LIN {X 0,Y 523.96,Z 722.024,A -85,B 0,C 180,E1 -4662.837,E2 -4662.837} C_VEL
LIN {X 0,Y 524.007,Z 722.026,A -85,B 0,C 180,E1 -4665.236,E2 -4665.236} C_VEL
LIN {X 0,Y 524.015,Z 722.018,A -85,B 0,C 180,E1 -4668.394,E2 -4668.394} C_VEL
LIN {X 0,Y 524.003,Z 722.019,A -85,B 0,C 180,E1 -4671.516,E2 -4671.516} C_VEL
LIN {X 0,Y 524.085,Z 722.007,A -85,B 0,C 180,E1 -4674.614,E2 -4674.614} C_VEL
LIN {X 0,Y 524.116,Z 722.011,A -85,B 0,C 180,E1 -4677.694,E2 -4677.694} C_VEL
LIN {X 0,Y 524.126,Z 722.001,A -85,B 0,C 180,E1 -4680.768,E2 -4680.768} C_VEL
LIN {X 0,Y 524.075,Z 722.005,A -85,B 0,C 180,E1 -4683.075,E2 -4683.075} C_VEL
LIN {X 0,Y 524.046,Z 722.017,A -85,B 0,C 180,E1 -4686.159,E2 -4686.159} C_VEL
LIN {X 0,Y 524.002,Z 722.022,A -85,B 0,C 180,E1 -4689.262,E2 -4689.262} C_VEL
LIN {X 0,Y 524.005,Z 722.021,A -85,B 0,C 180,E1 -4691.739,E2 -4691.739} C_VEL
LIN {X 0,Y 523.995,Z 722.019,A -85,B 0,C 180,E1 -4695.052,E2 -4695.052} C_VEL
LIN {X 0,Y 523.967,Z 722.031,A -85,B 0,C 180,E1 -4697.969,E2 -4697.969} C_VEL
LIN {X 0,Y 523.974,Z 722.02,A -85,B 0,C 180,E1 -4700.41,E2 -4700.41} C_VEL
LIN {X 0,Y 523.919,Z 722.028,A -85,B 0,C 180,E1 -4702.893,E2 -4702.893} C_VEL
LIN {X 0,Y 523.955,Z 722.027,A -85,B 0,C 180,E1 -4705.418,E2 -4705.418} C_VEL
LIN {X 0,Y 523.972,Z 722.031,A -85,B 0,C 180,E1 -4707.999,E2 -4707.999} C_VEL
LIN {X 0,Y 523.947,Z 722.026,A -85,B 0,C 180,E1 -4710.855,E2 -4710.855} C_VEL
LIN {X 0,Y 523.963,Z 722.028,A -85,B 0,C 180,E1 -4713.735,E2 -4713.735} C_VEL
LIN {X 0,Y 523.925,Z 722.029,A -85,B 0,C 180,E1 -4716.404,E2 -4716.404} C_VEL
LIN {X 0,Y 523.933,Z 722.012,A -85,B 0,C 180,E1 -4719.084,E2 -4719.084} C_VEL
LIN {X 0,Y 523.974,Z 722.017,A -85,B 0,C 180,E1 -4721.312,E2 -4721.312} C_VEL
LIN {X 0,Y 523.957,Z 722.031,A -85,B 0,C 180,E1 -4724.691,E2 -4724.691} C_VEL
LIN {X 0,Y 523.958,Z 722.023,A -85,B 0,C 180,E1 -4727.882,E2 -4727.882} C_VEL
LIN {X 0,Y 523.928,Z 722.034,A -85,B 0,C 180,E1 -4730.916,E2 -4730.916} C_VEL
LIN {X 0,Y 523.929,Z 722.027,A -85,B 0,C 180,E1 -4733.828,E2 -4733.828} C_VEL
LIN {X 0,Y 523.945,Z 722.036,A -85,B 0,C 180,E1 -4736.636,E2 -4736.636} C_VEL
LIN {X 0,Y 523.958,Z 722.022,A -85,B 0,C 180,E1 -4739.356,E2 -4739.356} C_VEL
LIN {X 0,Y 523.979,Z 722.027,A -85,B 0,C 180,E1 -4742.281,E2 -4742.281} C_VEL
LIN {X 0,Y 523.949,Z 722.033,A -85,B 0,C 180,E1 -4744.581,E2 -4744.581} C_VEL
LIN {X 0,Y 523.97,Z 722.172,A -85,B 0,C 180,E1 -4747.4,E2 -4747.4} C_VEL
LIN {X 0,Y 524.887,Z 728.251,A -85,B 0,C 180,E1 -4748.601,E2 -4748.601} C_VEL
LIN {X 0,Y 524.571,Z 744.644,A -85,B 0,C 180,E1 -4751.649,E2 -4751.649} C_VEL
LIN {X 0,Y 524.221,Z 761.458,A -85,B 0,C 180,E1 -4754.724,E2 -4754.724} C_VEL
LIN {X 0,Y 523.899,Z 779.887,A -85,B 0,C 180,E1 -4758.045,E2 -4758.045} C_VEL
LIN {X 0,Y 524.091,Z 781.846,A -85,B 0,C 180,E1 -4758.12,E2 -4758.12} C_VEL
LIN {X 0,Y 524.986,Z 790.156,A -85,B 0,C 180,E1 -4758.254,E2 -4758.254} C_VEL
LIN {X 0,Y 524.799,Z 856.138,A -85,B 0,C 180,E1 -4759.17,E2 -4759.17} C_VEL
LIN {X 0,Y 524.675,Z 865.409,A -85,B 0,C 180,E1 -4759.387,E2 -4759.387} C_VEL
LIN {X 0,Y 524.58,Z 873.883,A -85,B 0,C 180,E1 -4759.677,E2 -4759.677} C_VEL
LIN {X 0,Y 524.407,Z 882.388,A -85,B 0,C 180,E1 -4760.064,E2 -4760.064} C_VEL
LIN {X 0,Y 524.242,Z 890.722,A -85,B 0,C 180,E1 -4760.548,E2 -4760.548} C_VEL
LIN {X 0,Y 524.079,Z 898.761,A -85,B 0,C 180,E1 -4761.129,E2 -4761.129} C_VEL
LIN {X 0,Y 523.896,Z 907.432,A -85,B 0,C 180,E1 -4761.903,E2 -4761.903} C_VEL
LIN {X 0,Y 523.734,Z 915.938,A -85,B 0,C 180,E1 -4762.87,E2 -4762.87} C_VEL
LIN {X 0,Y 523.637,Z 922.61,A -85,B 0,C 180,E1 -4763.836,E2 -4763.836} C_VEL
LIN {X 0,Y 523.484,Z 926.989,A -85,B 0,C 180,E1 -4764.607,E2 -4764.607} C_VEL
LIN {X 0,Y 523.469,Z 932.149,A -85,B 0,C 180,E1 -4765.765,E2 -4765.765} C_VEL
LIN {X 0,Y 523.38,Z 935.937,A -85,B 0,C 180,E1 -4766.921,E2 -4766.921} C_VEL
LIN {X 0,Y 523.334,Z 937.681,A -85,B 0,C 180,E1 -4767.691,E2 -4767.691} C_VEL
LIN {X 0,Y 523.273,Z 938.93,A -85,B 0,C 180,E1 -4768.461,E2 -4768.461} C_VEL
LIN {X 0,Y 523.248,Z 939.707,A -85,B 0,C 180,E1 -4769.23,E2 -4769.23} C_VEL
LIN {X 0,Y 523.244,Z 940,A -85,B 0,C 180,E1 -4770,E2 -4770} C_VEL
LIN {X 0,Y 523.248,Z 939.707,A -85,B 0,C 180,E1 -4770.77,E2 -4770.77} C_VEL
LIN {X 0,Y 523.273,Z 938.929,A -85,B 0,C 180,E1 -4771.539,E2 -4771.539} C_VEL
LIN {X 0,Y 523.334,Z 937.68,A -85,B 0,C 180,E1 -4772.309,E2 -4772.309} C_VEL
LIN {X 0,Y 523.407,Z 934.786,A -85,B 0,C 180,E1 -4773.464,E2 -4773.464} C_VEL
LIN {X 0,Y 523.469,Z 932.149,A -85,B 0,C 180,E1 -4774.235,E2 -4774.235} C_VEL
LIN {X 0,Y 523.484,Z 926.986,A -85,B 0,C 180,E1 -4775.393,E2 -4775.393} C_VEL
LIN {X 0,Y 523.668,Z 920.738,A -85,B 0,C 180,E1 -4776.468,E2 -4776.468} C_VEL
LIN {X 0,Y 523.757,Z 912.74,A -85,B 0,C 180,E1 -4777.518,E2 -4777.518} C_VEL
LIN {X 0,Y 523.931,Z 905.398,A -85,B 0,C 180,E1 -4778.291,E2 -4778.291} C_VEL
LIN {X 0,Y 524.102,Z 897.534,A -85,B 0,C 180,E1 -4778.968,E2 -4778.968} C_VEL
LIN {X 0,Y 524.272,Z 889.222,A -85,B 0,C 180,E1 -4779.549,E2 -4779.549} C_VEL
LIN {X 0,Y 524.477,Z 878.61,A -85,B 0,C 180,E1 -4780.13,E2 -4780.13} C_VEL
LIN {X 0,Y 524.667,Z 867.075,A -85,B 0,C 180,E1 -4780.565,E2 -4780.565} C_VEL
LIN {X 0,Y 524.763,Z 857.437,A -85,B 0,C 180,E1 -4780.807,E2 -4780.807} C_VEL
LIN {X 0,Y 524.938,Z 807.339,A -85,B 0,C 180,E1 -4781.512,E2 -4781.512} C_VEL
LIN {X 0,Y 524.813,Z 787.359,A -85,B 0,C 180,E1 -4781.788,E2 -4781.788} C_VEL
LIN {X 0,Y 523.904,Z 780.121,A -85,B 0,C 180,E1 -4781.935,E2 -4781.935} C_VEL
LIN {X 0,Y 523.982,Z 772.996,A -85,B 0,C 180,E1 -4783.18,E2 -4783.18} C_VEL
LIN {X 0,Y 524.271,Z 757.745,A -85,B 0,C 180,E1 -4785.951,E2 -4785.951} C_VEL
LIN {X 0,Y 524.624,Z 741.367,A -85,B 0,C 180,E1 -4788.957,E2 -4788.957} C_VEL
LIN {X 0,Y 524.887,Z 728.251,A -85,B 0,C 180,E1 -4791.399,E2 -4791.399} C_VEL
LIN {X 0,Y 523.952,Z 722.075,A -85,B 0,C 180,E1 -4792.643,E2 -4792.643} C_VEL
LIN {X 0,Y 523.949,Z 722.033,A -85,B 0,C 180,E1 -4795.419,E2 -4795.419} C_VEL
LIN {X 0,Y 523.97,Z 722.026,A -85,B 0,C 180,E1 -4797.999,E2 -4797.999} C_VEL
LIN {X 0,Y 523.948,Z 722.024,A -85,B 0,C 180,E1 -4800.855,E2 -4800.855} C_VEL
LIN {X 0,Y 523.963,Z 722.03,A -85,B 0,C 180,E1 -4803.735,E2 -4803.735} C_VEL
LIN {X 0,Y 523.924,Z 722.028,A -85,B 0,C 180,E1 -4806.404,E2 -4806.404} C_VEL
LIN {X 0,Y 523.928,Z 722.033,A -85,B 0,C 180,E1 -4809.084,E2 -4809.084} C_VEL
LIN {X 0,Y 523.958,Z 722.024,A -85,B 0,C 180,E1 -4812.118,E2 -4812.118} C_VEL
LIN {X 0,Y 523.957,Z 722.031,A -85,B 0,C 180,E1 -4815.309,E2 -4815.309} C_VEL
LIN {X 0,Y 523.974,Z 722.016,A -85,B 0,C 180,E1 -4818.688,E2 -4818.688} C_VEL
LIN {X 0,Y 523.927,Z 722.013,A -85,B 0,C 180,E1 -4821.079,E2 -4821.079} C_VEL
LIN {X 0,Y 523.93,Z 722.033,A -85,B 0,C 180,E1 -4823.828,E2 -4823.828} C_VEL
LIN {X 0,Y 523.944,Z 722.028,A -85,B 0,C 180,E1 -4826.636,E2 -4826.636} C_VEL
LIN {X 0,Y 523.958,Z 722.026,A -85,B 0,C 180,E1 -4829.356,E2 -4829.356} C_VEL
LIN {X 0,Y 523.981,Z 722.026,A -85,B 0,C 180,E1 -4832.281,E2 -4832.281} C_VEL
LIN {X 0,Y 523.955,Z 722.027,A -85,B 0,C 180,E1 -4834.582,E2 -4834.582} C_VEL
LIN {X 0,Y 523.919,Z 722.027,A -85,B 0,C 180,E1 -4837.107,E2 -4837.107} C_VEL
LIN {X 0,Y 523.981,Z 722.023,A -85,B 0,C 180,E1 -4839.866,E2 -4839.866} C_VEL
LIN {X 0,Y 523.973,Z 722.024,A -85,B 0,C 180,E1 -4842.838,E2 -4842.838} C_VEL
LIN {X 0,Y 523.979,Z 722.021,A -85,B 0,C 180,E1 -4845.236,E2 -4845.236} C_VEL
LIN {X 0,Y 524.015,Z 722.021,A -85,B 0,C 180,E1 -4848.394,E2 -4848.394} C_VEL
LIN {X 0,Y 524.007,Z 722.019,A -85,B 0,C 180,E1 -4851.516,E2 -4851.516} C_VEL
LIN {X 0,Y 524.084,Z 722.013,A -85,B 0,C 180,E1 -4854.614,E2 -4854.614} C_VEL
LIN {X 0,Y 524.114,Z 721.998,A -85,B 0,C 180,E1 -4857.695,E2 -4857.695} C_VEL
LIN {X 0,Y 524.126,Z 722.01,A -85,B 0,C 180,E1 -4860.768,E2 -4860.768} C_VEL
LIN {X 0,Y 524.075,Z 722.013,A -85,B 0,C 180,E1 -4863.075,E2 -4863.075} C_VEL
LIN {X 0,Y 524.04,Z 722.015,A -85,B 0,C 180,E1 -4866.159,E2 -4866.159} C_VEL
LIN {X 0,Y 524.003,Z 722.018,A -85,B 0,C 180,E1 -4868.484,E2 -4868.484} C_VEL
LIN {X 0,Y 524.006,Z 722.019,A -85,B 0,C 180,E1 -4871.74,E2 -4871.74} C_VEL
LIN {X 0,Y 523.996,Z 722.023,A -85,B 0,C 180,E1 -4875.052,E2 -4875.052} C_VEL
LIN {X 0,Y 523.95,Z 722.021,A -85,B 0,C 180,E1 -4877.97,E2 -4877.97} C_VEL
LIN {X 0,Y 523.974,Z 722.024,A -85,B 0,C 180,E1 -4880.41,E2 -4880.41} C_VEL
LIN {X 0,Y 523.912,Z 722.04,A -85,B 0,C 180,E1 -4882.894,E2 -4882.894} C_VEL
LIN {X 0,Y 523.985,Z 722.016,A -85,B 0,C 180,E1 -4886.019,E2 -4886.019} C_VEL
LIN {X 0,Y 523.937,Z 722.033,A -85,B 0,C 180,E1 -4888.875,E2 -4888.875} C_VEL
LIN {X 0,Y 523.921,Z 722.032,A -85,B 0,C 180,E1 -4891.544,E2 -4891.544} C_VEL
LIN {X 0,Y 523.922,Z 722.027,A -85,B 0,C 180,E1 -4894.291,E2 -4894.291} C_VEL
LIN {X 0,Y 523.908,Z 722.039,A -85,B 0,C 180,E1 -4897.132,E2 -4897.132} C_VEL
LIN {X 0,Y 523.939,Z 722.023,A -85,B 0,C 180,E1 -4900.13,E2 -4900.13} C_VEL
LIN {X 0,Y 523.933,Z 722.013,A -85,B 0,C 180,E1 -4902.458,E2 -4902.458} C_VEL
LIN {X 0,Y 523.944,Z 722.029,A -85,B 0,C 180,E1 -4905.31,E2 -4905.31} C_VEL
LIN {X 0,Y 523.916,Z 722.032,A -85,B 0,C 180,E1 -4906.909,E2 -4906.909} C_VEL
LIN {X 0,Y 523.252,Z 722.122,A -85,B 0,C 180,E1 -4907.55,E2 -4907.55} C_VEL
LIN {X 0,Y 520.412,Z 722.471,A -85,B 0,C 180,E1 -4908.592,E2 -4908.592} C_VEL
LIN {X 0,Y 518.007,Z 722.774,A -85,B 0,C 180,E1 -4909.431,E2 -4909.431} C_VEL
LIN {X 0,Y 516.97,Z 722.894,A -85,B 0,C 180,E1 -4910.079,E2 -4910.079} C_VEL
LIN {X 0,Y 516.883,Z 722.903,A -85,B 0,C 180,E1 -4910.298,E2 -4910.298} C_VEL
LIN {X 0,Y 516.878,Z 722.909,A -85,B 0,C 180,E1 -4913.343,E2 -4913.343} C_VEL
LIN {X 0,Y 516.885,Z 722.909,A -85,B 0,C 180,E1 -4916.119,E2 -4916.119} C_VEL
LIN {X 0,Y 516.891,Z 722.903,A -85,B 0,C 180,E1 -4918.936,E2 -4918.936} C_VEL
LIN {X 0,Y 516.864,Z 722.917,A -85,B 0,C 180,E1 -4921.581,E2 -4921.581} C_VEL
LIN {X 0,Y 516.885,Z 722.911,A -85,B 0,C 180,E1 -4924.208,E2 -4924.208} C_VEL
LIN {X 0,Y 516.86,Z 722.909,A -85,B 0,C 180,E1 -4926.776,E2 -4926.776} C_VEL
LIN {X 0,Y 516.941,Z 722.908,A -85,B 0,C 180,E1 -4929.732,E2 -4929.732} C_VEL
LIN {X 0,Y 517.031,Z 723.121,A -85,B 0,C 180,E1 -4931.32,E2 -4931.32} C_VEL
LIN {X 0,Y 517.103,Z 730.186,A -85,B 0,C 180,E1 -4933.01,E2 -4933.01} C_VEL
LIN {X 0,Y 516.819,Z 742.298,A -85,B 0,C 180,E1 -4935.831,E2 -4935.831} C_VEL
LIN {X 0,Y 516.707,Z 751.608,A -85,B 0,C 180,E1 -4937.94,E2 -4937.94} C_VEL
LIN {X 0,Y 517.044,Z 754.054,A -85,B 0,C 180,E1 -4938.029,E2 -4938.029} C_VEL
LIN {X 0,Y 518.001,Z 762.348,A -85,B 0,C 180,E1 -4938.167,E2 -4938.167} C_VEL
LIN {X 0,Y 517.785,Z 826.462,A -85,B 0,C 180,E1 -4939.07,E2 -4939.07} C_VEL
LIN {X 0,Y 517.706,Z 835.644,A -85,B 0,C 180,E1 -4939.292,E2 -4939.292} C_VEL
LIN {X 0,Y 517.546,Z 845.274,A -85,B 0,C 180,E1 -4939.634,E2 -4939.634} C_VEL
LIN {X 0,Y 517.414,Z 855.328,A -85,B 0,C 180,E1 -4940.126,E2 -4940.126} C_VEL
LIN {X 0,Y 517.184,Z 865.799,A -85,B 0,C 180,E1 -4940.812,E2 -4940.812} C_VEL
LIN {X 0,Y 516.898,Z 875.032,A -85,B 0,C 180,E1 -4941.595,E2 -4941.595} C_VEL
LIN {X 0,Y 516.703,Z 882.414,A -85,B 0,C 180,E1 -4942.379,E2 -4942.379} C_VEL
LIN {X 0,Y 516.597,Z 889.273,A -85,B 0,C 180,E1 -4943.277,E2 -4943.277} C_VEL
LIN {X 0,Y 516.499,Z 895.801,A -85,B 0,C 180,E1 -4944.339,E2 -4944.339} C_VEL
LIN {X 0,Y 516.322,Z 900.458,A -85,B 0,C 180,E1 -4945.315,E2 -4945.315} C_VEL
LIN {X 0,Y 516.385,Z 903.47,A -85,B 0,C 180,E1 -4946.098,E2 -4946.098} C_VEL
LIN {X 0,Y 516.295,Z 905.809,A -85,B 0,C 180,E1 -4946.879,E2 -4946.879} C_VEL
LIN {X 0,Y 516.263,Z 907.59,A -85,B 0,C 180,E1 -4947.659,E2 -4947.659} C_VEL
LIN {X 0,Y 516.19,Z 908.875,A -85,B 0,C 180,E1 -4948.44,E2 -4948.44} C_VEL
LIN {X 0,Y 516.157,Z 909.689,A -85,B 0,C 180,E1 -4949.22,E2 -4949.22} C_VEL
LIN {X 0,Y 516.152,Z 909.997,A -85,B 0,C 180,E1 -4950,E2 -4950} C_VEL
LIN {X 0,Y 516.157,Z 909.726,A -85,B 0,C 180,E1 -4950.78,E2 -4950.78} C_VEL
LIN {X 0,Y 516.191,Z 908.986,A -85,B 0,C 180,E1 -4951.56,E2 -4951.56} C_VEL
LIN {X 0,Y 516.263,Z 907.777,A -85,B 0,C 180,E1 -4952.341,E2 -4952.341} C_VEL
LIN {X 0,Y 516.324,Z 904.921,A -85,B 0,C 180,E1 -4953.512,E2 -4953.512} C_VEL
LIN {X 0,Y 516.39,Z 902.325,A -85,B 0,C 180,E1 -4954.293,E2 -4954.293} C_VEL
LIN {X 0,Y 516.431,Z 897.208,A -85,B 0,C 180,E1 -4955.466,E2 -4955.466} C_VEL
LIN {X 0,Y 516.59,Z 891.595,A -85,B 0,C 180,E1 -4956.462,E2 -4956.462} C_VEL
LIN {X 0,Y 516.691,Z 883.161,A -85,B 0,C 180,E1 -4957.621,E2 -4957.621} C_VEL
LIN {X 0,Y 516.916,Z 874.939,A -85,B 0,C 180,E1 -4958.503,E2 -4958.503} C_VEL
LIN {X 0,Y 517.157,Z 865.674,A -85,B 0,C 180,E1 -4959.287,E2 -4959.287} C_VEL
LIN {X 0,Y 517.369,Z 855.163,A -85,B 0,C 180,E1 -4959.974,E2 -4959.974} C_VEL
LIN {X 0,Y 517.578,Z 845.055,A -85,B 0,C 180,E1 -4960.464,E2 -4960.464} C_VEL
LIN {X 0,Y 517.691,Z 836.176,A -85,B 0,C 180,E1 -4960.783,E2 -4960.783} C_VEL
LIN {X 0,Y 517.845,Z 827.357,A -85,B 0,C 180,E1 -4961.001,E2 -4961.001} C_VEL
LIN {X 0,Y 517.932,Z 760.029,A -85,B 0,C 180,E1 -4961.957,E2 -4961.957} C_VEL
LIN {X 0,Y 516.695,Z 751.778,A -85,B 0,C 180,E1 -4962.126,E2 -4962.126} C_VEL
LIN {X 0,Y 516.647,Z 751.291,A -85,B 0,C 180,E1 -4962.172,E2 -4962.172} C_VEL
LIN {X 0,Y 516.952,Z 737.395,A -85,B 0,C 180,E1 -4965.394,E2 -4965.394} C_VEL
LIN {X 0,Y 517.152,Z 725.401,A -85,B 0,C 180,E1 -4968.214,E2 -4968.214} C_VEL
LIN {X 0,Y 516.985,Z 722.989,A -85,B 0,C 180,E1 -4968.836,E2 -4968.836} C_VEL
LIN {X 0,Y 516.887,Z 722.909,A -85,B 0,C 180,E1 -4971.538,E2 -4971.538} C_VEL
LIN {X 0,Y 516.876,Z 722.917,A -85,B 0,C 180,E1 -4974.355,E2 -4974.355} C_VEL
LIN {X 0,Y 516.892,Z 722.907,A -85,B 0,C 180,E1 -4977.535,E2 -4977.535} C_VEL
LIN {X 0,Y 516.888,Z 722.914,A -85,B 0,C 180,E1 -4980.204,E2 -4980.204} C_VEL
LIN {X 0,Y 516.882,Z 722.909,A -85,B 0,C 180,E1 -4982.948,E2 -4982.948} C_VEL
LIN {X 0,Y 516.872,Z 722.911,A -85,B 0,C 180,E1 -4985.78,E2 -4985.78} C_VEL
LIN {X 0,Y 516.879,Z 722.908,A -85,B 0,C 180,E1 -4988.716,E2 -4988.716} C_VEL
LIN {X 0,Y 516.913,Z 722.903,A -85,B 0,C 180,E1 -4991.775,E2 -4991.775} C_VEL
LIN {X 0,Y 516.896,Z 722.903,A -85,B 0,C 180,E1 -4995.007,E2 -4995.007} C_VEL
LIN {X 0,Y 516.914,Z 722.891,A -85,B 0,C 180,E1 -4998.399,E2 -4998.399} C_VEL
LIN {X 0,Y 516.88,Z 722.908,A -85,B 0,C 180,E1 -5001.284,E2 -5001.284} C_VEL
LIN {X 0,Y 516.872,Z 722.91,A -85,B 0,C 180,E1 -5004.22,E2 -5004.22} C_VEL
LIN {X 0,Y 516.883,Z 722.911,A -85,B 0,C 180,E1 -5007.052,E2 -5007.052} C_VEL
LIN {X 0,Y 516.888,Z 722.906,A -85,B 0,C 180,E1 -5009.796,E2 -5009.796} C_VEL
LIN {X 0,Y 516.926,Z 722.903,A -85,B 0,C 180,E1 -5012.467,E2 -5012.467} C_VEL
LIN {X 0,Y 516.908,Z 722.907,A -85,B 0,C 180,E1 -5015.072,E2 -5015.072} C_VEL
LIN {X 0,Y 516.888,Z 722.907,A -85,B 0,C 180,E1 -5018.462,E2 -5018.462} C_VEL
LIN {X 0,Y 516.903,Z 722.91,A -85,B 0,C 180,E1 -5020.955,E2 -5020.955} C_VEL
LIN {X 0,Y 516.911,Z 722.905,A -85,B 0,C 180,E1 -5023.41,E2 -5023.41} C_VEL
LIN {X 0,Y 516.907,Z 722.905,A -85,B 0,C 180,E1 -5025.834,E2 -5025.834} C_VEL
LIN {X 0,Y 516.954,Z 722.903,A -85,B 0,C 180,E1 -5029.028,E2 -5029.028} C_VEL
LIN {X 0,Y 516.98,Z 722.886,A -85,B 0,C 180,E1 -5032.187,E2 -5032.187} C_VEL
LIN {X 0,Y 517.031,Z 722.885,A -85,B 0,C 180,E1 -5034.54,E2 -5034.54} C_VEL
LIN {X 0,Y 517.088,Z 722.887,A -85,B 0,C 180,E1 -5037.663,E2 -5037.663} C_VEL
LIN {X 0,Y 517.096,Z 722.877,A -85,B 0,C 180,E1 -5040.779,E2 -5040.779} C_VEL
LIN {X 0,Y 517.015,Z 722.884,A -85,B 0,C 180,E1 -5043.117,E2 -5043.117} C_VEL
LIN {X 0,Y 517.011,Z 722.892,A -85,B 0,C 180,E1 -5046.243,E2 -5046.243} C_VEL
LIN {X 0,Y 516.956,Z 722.902,A -85,B 0,C 180,E1 -5049.389,E2 -5049.389} C_VEL
LIN {X 0,Y 516.954,Z 722.898,A -85,B 0,C 180,E1 -5051.807,E2 -5051.807} C_VEL
LIN {X 0,Y 516.947,Z 722.898,A -85,B 0,C 180,E1 -5055.146,E2 -5055.146} C_VEL
LIN {X 0,Y 516.928,Z 722.904,A -85,B 0,C 180,E1 -5058.222,E2 -5058.222} C_VEL
LIN {X 0,Y 516.915,Z 722.897,A -85,B 0,C 180,E1 -5060.701,E2 -5060.701} C_VEL
LIN {X 0,Y 516.913,Z 722.912,A -85,B 0,C 180,E1 -5064.072,E2 -5064.072} C_VEL
LIN {X 0,Y 516.928,Z 722.902,A -85,B 0,C 180,E1 -5066.658,E2 -5066.658} C_VEL
LIN {X 0,Y 516.913,Z 722.899,A -85,B 0,C 180,E1 -5069.524,E2 -5069.524} C_VEL
LIN {X 0,Y 516.899,Z 722.909,A -85,B 0,C 180,E1 -5072.544,E2 -5072.544} C_VEL
LIN {X 0,Y 516.885,Z 722.905,A -85,B 0,C 180,E1 -5075.332,E2 -5075.332} C_VEL
LIN {X 0,Y 516.883,Z 722.903,A -85,B 0,C 180,E1 -5077.943,E2 -5077.943} C_VEL
LIN {X 0,Y 516.905,Z 722.9,A -85,B 0,C 180,E1 -5080.739,E2 -5080.739} C_VEL
LIN {X 0,Y 516.884,Z 722.908,A -85,B 0,C 180,E1 -5083.903,E2 -5083.903} C_VEL
LIN {X 0,Y 516.883,Z 722.911,A -85,B 0,C 180,E1 -5086.107,E2 -5086.107} C_VEL
LIN {X 0,Y 516.918,Z 722.904,A -85,B 0,C 180,E1 -5088.398,E2 -5088.398} C_VEL
LIN {X 0,Y 516.886,Z 722.908,A -85,B 0,C 180,E1 -5091.284,E2 -5091.284} C_VEL
LIN {X 0,Y 516.892,Z 722.907,A -85,B 0,C 180,E1 -5094.221,E2 -5094.221} C_VEL
LIN {X 0,Y 516.899,Z 722.907,A -85,B 0,C 180,E1 -5097.053,E2 -5097.053} C_VEL
LIN {X 0,Y 516.894,Z 722.9,A -85,B 0,C 180,E1 -5099.796,E2 -5099.796} C_VEL
LIN {X 0,Y 516.929,Z 722.908,A -85,B 0,C 180,E1 -5102.467,E2 -5102.467} C_VEL
LIN {X 0,Y 516.905,Z 722.909,A -85,B 0,C 180,E1 -5105.072,E2 -5105.072} C_VEL
LIN {X 0,Y 516.908,Z 723.029,A -85,B 0,C 180,E1 -5107.26,E2 -5107.26} C_VEL
LIN {X 0,Y 517.89,Z 729.171,A -85,B 0,C 180,E1 -5108.506,E2 -5108.506} C_VEL
LIN {X 0,Y 517.556,Z 745.565,A -85,B 0,C 180,E1 -5111.596,E2 -5111.596} C_VEL
LIN {X 0,Y 517.158,Z 762.669,A -85,B 0,C 180,E1 -5114.767,E2 -5114.767} C_VEL
LIN {X 0,Y 516.825,Z 779.847,A -85,B 0,C 180,E1 -5117.883,E2 -5117.883} C_VEL
LIN {X 0,Y 517.051,Z 781.622,A -85,B 0,C 180,E1 -5117.954,E2 -5117.954} C_VEL
LIN {X 0,Y 518.035,Z 790.103,A -85,B 0,C 180,E1 -5118.094,E2 -5118.094} C_VEL
LIN {X 0,Y 517.842,Z 856.135,A -85,B 0,C 180,E1 -5119.022,E2 -5119.022} C_VEL
LIN {X 0,Y 517.684,Z 865.407,A -85,B 0,C 180,E1 -5119.242,E2 -5119.242} C_VEL
LIN {X 0,Y 517.604,Z 873.881,A -85,B 0,C 180,E1 -5119.537,E2 -5119.537} C_VEL
LIN {X 0,Y 517.419,Z 882.386,A -85,B 0,C 180,E1 -5119.928,E2 -5119.928} C_VEL
LIN {X 0,Y 517.249,Z 890.72,A -85,B 0,C 180,E1 -5120.419,E2 -5120.419} C_VEL
LIN {X 0,Y 517.068,Z 898.758,A -85,B 0,C 180,E1 -5121.007,E2 -5121.007} C_VEL
LIN {X 0,Y 516.847,Z 907.431,A -85,B 0,C 180,E1 -5121.791,E2 -5121.791} C_VEL
LIN {X 0,Y 516.692,Z 915.938,A -85,B 0,C 180,E1 -5122.772,E2 -5122.772} C_VEL
LIN {X 0,Y 516.571,Z 922.609,A -85,B 0,C 180,E1 -5123.751,E2 -5123.751} C_VEL
LIN {X 0,Y 516.431,Z 926.989,A -85,B 0,C 180,E1 -5124.534,E2 -5124.534} C_VEL
LIN {X 0,Y 516.392,Z 932.149,A -85,B 0,C 180,E1 -5125.707,E2 -5125.707} C_VEL
LIN {X 0,Y 516.325,Z 934.787,A -85,B 0,C 180,E1 -5126.488,E2 -5126.488} C_VEL
LIN {X 0,Y 516.261,Z 937.68,A -85,B 0,C 180,E1 -5127.659,E2 -5127.659} C_VEL
LIN {X 0,Y 516.19,Z 938.929,A -85,B 0,C 180,E1 -5128.44,E2 -5128.44} C_VEL
LIN {X 0,Y 516.158,Z 939.706,A -85,B 0,C 180,E1 -5129.22,E2 -5129.22} C_VEL
LIN {X 0,Y 516.151,Z 940,A -85,B 0,C 180,E1 -5130,E2 -5130} C_VEL
LIN {X 0,Y 516.158,Z 939.706,A -85,B 0,C 180,E1 -5130.78,E2 -5130.78} C_VEL
LIN {X 0,Y 516.19,Z 938.928,A -85,B 0,C 180,E1 -5131.56,E2 -5131.56} C_VEL
LIN {X 0,Y 516.261,Z 937.679,A -85,B 0,C 180,E1 -5132.341,E2 -5132.341} C_VEL
LIN {X 0,Y 516.325,Z 934.786,A -85,B 0,C 180,E1 -5133.512,E2 -5133.512} C_VEL
LIN {X 0,Y 516.392,Z 932.149,A -85,B 0,C 180,E1 -5134.293,E2 -5134.293} C_VEL
LIN {X 0,Y 516.431,Z 926.985,A -85,B 0,C 180,E1 -5135.466,E2 -5135.466} C_VEL
LIN {X 0,Y 516.58,Z 921.233,A -85,B 0,C 180,E1 -5136.478,E2 -5136.478} C_VEL
LIN {X 0,Y 516.686,Z 914.435,A -85,B 0,C 180,E1 -5137.425,E2 -5137.425} C_VEL
LIN {X 0,Y 516.863,Z 906.418,A -85,B 0,C 180,E1 -5138.307,E2 -5138.307} C_VEL
LIN {X 0,Y 517.068,Z 898.763,A -85,B 0,C 180,E1 -5138.993,E2 -5138.993} C_VEL
LIN {X 0,Y 517.249,Z 890.721,A -85,B 0,C 180,E1 -5139.581,E2 -5139.581} C_VEL
LIN {X 0,Y 517.419,Z 882.388,A -85,B 0,C 180,E1 -5140.072,E2 -5140.072} C_VEL
LIN {X 0,Y 517.614,Z 873.885,A -85,B 0,C 180,E1 -5140.463,E2 -5140.463} C_VEL
LIN {X 0,Y 517.71,Z 863.745,A -85,B 0,C 180,E1 -5140.807,E2 -5140.807} C_VEL
LIN {X 0,Y 517.912,Z 852.082,A -85,B 0,C 180,E1 -5141.05,E2 -5141.05} C_VEL
LIN {X 0,Y 517.876,Z 787.906,A -85,B 0,C 180,E1 -5141.94,E2 -5141.94} C_VEL
LIN {X 0,Y 516.843,Z 780.138,A -85,B 0,C 180,E1 -5142.094,E2 -5142.094} C_VEL
LIN {X 0,Y 516.863,Z 777.221,A -85,B 0,C 180,E1 -5142.566,E2 -5142.566} C_VEL
LIN {X 0,Y 517.174,Z 761.553,A -85,B 0,C 180,E1 -5145.437,E2 -5145.437} C_VEL
LIN {X 0,Y 517.556,Z 745.56,A -85,B 0,C 180,E1 -5148.404,E2 -5148.404} C_VEL
LIN {X 0,Y 517.912,Z 730.264,A -85,B 0,C 180,E1 -5151.284,E2 -5151.284} C_VEL
LIN {X 0,Y 517.164,Z 724.233,A -85,B 0,C 180,E1 -5152.469,E2 -5152.469} C_VEL
LIN {X 0,Y 516.905,Z 722.934,A -85,B 0,C 180,E1 -5152.798,E2 -5152.798} C_VEL
LIN {X 0,Y 516.944,Z 722.899,A -85,B 0,C 180,E1 -5156.196,E2 -5156.196} C_VEL
LIN {X 0,Y 516.923,Z 722.906,A -85,B 0,C 180,E1 -5159.304,E2 -5159.304} C_VEL
LIN {X 0,Y 516.902,Z 722.904,A -85,B 0,C 180,E1 -5162.544,E2 -5162.544} C_VEL
LIN {X 0,Y 516.884,Z 722.913,A -85,B 0,C 180,E1 -5165.333,E2 -5165.333} C_VEL
LIN {X 0,Y 516.883,Z 722.91,A -85,B 0,C 180,E1 -5167.943,E2 -5167.943} C_VEL
LIN {X 0,Y 516.887,Z 722.903,A -85,B 0,C 180,E1 -5170.741,E2 -5170.741} C_VEL
LIN {X 0,Y 516.885,Z 722.904,A -85,B 0,C 180,E1 -5172.831,E2 -5172.831} C_VEL
LIN {X 0,Y 516.924,Z 722.904,A -85,B 0,C 180,E1 -5175.01,E2 -5175.01} C_VEL
LIN {X 0,Y 516.924,Z 722.895,A -85,B 0,C 180,E1 -5178.398,E2 -5178.398} C_VEL
LIN {X 0,Y 516.888,Z 722.89,A -85,B 0,C 180,E1 -5181.285,E2 -5181.285} C_VEL
LIN {X 0,Y 516.893,Z 722.907,A -85,B 0,C 180,E1 -5184.221,E2 -5184.221} C_VEL
LIN {X 0,Y 516.898,Z 722.906,A -85,B 0,C 180,E1 -5187.053,E2 -5187.053} C_VEL
LIN {X 0,Y 516.894,Z 722.91,A -85,B 0,C 180,E1 -5189.797,E2 -5189.797} C_VEL
LIN {X 0,Y 516.93,Z 722.903,A -85,B 0,C 180,E1 -5192.468,E2 -5192.468} C_VEL
LIN {X 0,Y 516.913,Z 722.903,A -85,B 0,C 180,E1 -5195.072,E2 -5195.072} C_VEL
LIN {X 0,Y 516.872,Z 722.908,A -85,B 0,C 180,E1 -5197.622,E2 -5197.622} C_VEL
LIN {X 0,Y 516.935,Z 722.905,A -85,B 0,C 180,E1 -5200.13,E2 -5200.13} C_VEL
LIN {X 0,Y 516.933,Z 722.904,A -85,B 0,C 180,E1 -5202.596,E2 -5202.596} C_VEL
LIN {X 0,Y 516.944,Z 722.897,A -85,B 0,C 180,E1 -5205.03,E2 -5205.03} C_VEL
LIN {X 0,Y 516.968,Z 722.897,A -85,B 0,C 180,E1 -5208.234,E2 -5208.234} C_VEL
LIN {X 0,Y 516.972,Z 722.895,A -85,B 0,C 180,E1 -5211.4,E2 -5211.4} C_VEL
LIN {X 0,Y 517.011,Z 722.892,A -85,B 0,C 180,E1 -5213.757,E2 -5213.757} C_VEL
LIN {X 0,Y 517.087,Z 722.873,A -85,B 0,C 180,E1 -5217.663,E2 -5217.663} C_VEL
LIN {X 0,Y 517.096,Z 722.885,A -85,B 0,C 180,E1 -5220.779,E2 -5220.779} C_VEL
LIN {X 0,Y 517.016,Z 722.892,A -85,B 0,C 180,E1 -5223.117,E2 -5223.117} C_VEL
LIN {X 0,Y 517.005,Z 722.892,A -85,B 0,C 180,E1 -5226.243,E2 -5226.243} C_VEL
LIN {X 0,Y 516.948,Z 722.897,A -85,B 0,C 180,E1 -5229.389,E2 -5229.389} C_VEL
LIN {X 0,Y 516.955,Z 722.898,A -85,B 0,C 180,E1 -5231.807,E2 -5231.807} C_VEL
LIN {X 0,Y 516.947,Z 722.899,A -85,B 0,C 180,E1 -5235.147,E2 -5235.147} C_VEL
LIN {X 0,Y 516.918,Z 722.897,A -85,B 0,C 180,E1 -5238.223,E2 -5238.223} C_VEL
LIN {X 0,Y 516.915,Z 722.907,A -85,B 0,C 180,E1 -5240.701,E2 -5240.701} C_VEL
LIN {X 0,Y 516.892,Z 722.904,A -85,B 0,C 180,E1 -5244.073,E2 -5244.073} C_VEL
LIN {X 0,Y 516.926,Z 722.898,A -85,B 0,C 180,E1 -5246.658,E2 -5246.658} C_VEL
LIN {X 0,Y 516.911,Z 722.907,A -85,B 0,C 180,E1 -5249.523,E2 -5249.523} C_VEL
LIN {X 0,Y 516.896,Z 722.904,A -85,B 0,C 180,E1 -5252.543,E2 -5252.543} C_VEL
LIN {X 0,Y 516.867,Z 722.917,A -85,B 0,C 180,E1 -5255.33,E2 -5255.33} C_VEL
LIN {X 0,Y 516.88,Z 722.907,A -85,B 0,C 180,E1 -5257.943,E2 -5257.943} C_VEL
LIN {X 0,Y 516.885,Z 722.902,A -85,B 0,C 180,E1 -5260.742,E2 -5260.742} C_VEL
LIN {X 0,Y 516.864,Z 722.894,A -85,B 0,C 180,E1 -5262.834,E2 -5262.834} C_VEL
LIN {X 0,Y 516.896,Z 722.902,A -85,B 0,C 180,E1 -5265.007,E2 -5265.007} C_VEL
LIN {X 0,Y 516.914,Z 722.903,A -85,B 0,C 180,E1 -5268.399,E2 -5268.399} C_VEL
LIN {X 0,Y 516.883,Z 722.903,A -85,B 0,C 180,E1 -5270.298,E2 -5270.298} C_VEL
LIN {X 0,Y 516.211,Z 722.988,A -85,B 0,C 180,E1 -5270.948,E2 -5270.948} C_VEL
LIN {X 0,Y 513.364,Z 723.349,A -85,B 0,C 180,E1 -5272.004,E2 -5272.004} C_VEL
LIN {X 0,Y 510.955,Z 723.654,A -85,B 0,C 180,E1 -5272.854,E2 -5272.854} C_VEL
LIN {X 0,Y 509.912,Z 723.782,A -85,B 0,C 180,E1 -5273.51,E2 -5273.51} C_VEL
LIN {X 0,Y 509.822,Z 723.792,A -85,B 0,C 180,E1 -5273.733,E2 -5273.733} C_VEL
LIN {X 0,Y 509.843,Z 723.784,A -85,B 0,C 180,E1 -5276.538,E2 -5276.538} C_VEL
LIN {X 0,Y 509.844,Z 723.784,A -85,B 0,C 180,E1 -5279.334,E2 -5279.334} C_VEL
LIN {X 0,Y 509.849,Z 723.789,A -85,B 0,C 180,E1 -5282.052,E2 -5282.052} C_VEL
LIN {X 0,Y 509.813,Z 723.789,A -85,B 0,C 180,E1 -5284.701,E2 -5284.701} C_VEL
LIN {X 0,Y 509.827,Z 723.789,A -85,B 0,C 180,E1 -5287.458,E2 -5287.458} C_VEL
LIN {X 0,Y 509.893,Z 723.786,A -85,B 0,C 180,E1 -5290.683,E2 -5290.683} C_VEL
LIN {X 0,Y 509.996,Z 723.933,A -85,B 0,C 180,E1 -5291.209,E2 -5291.209} C_VEL
LIN {X 0,Y 510.117,Z 730.352,A -85,B 0,C 180,E1 -5292.77,E2 -5292.77} C_VEL
LIN {X 0,Y 509.817,Z 742.464,A -85,B 0,C 180,E1 -5295.633,E2 -5295.633} C_VEL
LIN {X 0,Y 509.675,Z 751.798,A -85,B 0,C 180,E1 -5297.771,E2 -5297.771} C_VEL
LIN {X 0,Y 510.018,Z 754.22,A -85,B 0,C 180,E1 -5297.86,E2 -5297.86} C_VEL
LIN {X 0,Y 511.07,Z 762.602,A -85,B 0,C 180,E1 -5298.005,E2 -5298.005} C_VEL
LIN {X 0,Y 510.838,Z 826.703,A -85,B 0,C 180,E1 -5298.92,E2 -5298.92} C_VEL
LIN {X 0,Y 510.757,Z 835.873,A -85,B 0,C 180,E1 -5299.144,E2 -5299.144} C_VEL
LIN {X 0,Y 510.571,Z 845.496,A -85,B 0,C 180,E1 -5299.491,E2 -5299.491} C_VEL
LIN {X 0,Y 510.423,Z 855.546,A -85,B 0,C 180,E1 -5299.989,E2 -5299.989} C_VEL
LIN {X 0,Y 510.183,Z 865.972,A -85,B 0,C 180,E1 -5300.685,E2 -5300.685} C_VEL
LIN {X 0,Y 509.923,Z 874.121,A -85,B 0,C 180,E1 -5301.38,E2 -5301.38} C_VEL
LIN {X 0,Y 509.713,Z 880.841,A -85,B 0,C 180,E1 -5302.075,E2 -5302.075} C_VEL
LIN {X 0,Y 509.609,Z 887.199,A -85,B 0,C 180,E1 -5302.87,E2 -5302.87} C_VEL
LIN {X 0,Y 509.522,Z 892.483,A -85,B 0,C 180,E1 -5303.665,E2 -5303.665} C_VEL
LIN {X 0,Y 509.385,Z 896.896,A -85,B 0,C 180,E1 -5304.458,E2 -5304.458} C_VEL
LIN {X 0,Y 509.235,Z 900.571,A -85,B 0,C 180,E1 -5305.25,E2 -5305.25} C_VEL
LIN {X 0,Y 509.318,Z 903.564,A -85,B 0,C 180,E1 -5306.044,E2 -5306.044} C_VEL
LIN {X 0,Y 509.213,Z 905.893,A -85,B 0,C 180,E1 -5306.835,E2 -5306.835} C_VEL
LIN {X 0,Y 509.192,Z 907.664,A -85,B 0,C 180,E1 -5307.627,E2 -5307.627} C_VEL
LIN {X 0,Y 509.111,Z 908.944,A -85,B 0,C 180,E1 -5308.418,E2 -5308.418} C_VEL
LIN {X 0,Y 509.07,Z 909.754,A -85,B 0,C 180,E1 -5309.209,E2 -5309.209} C_VEL
LIN {X 0,Y 509.063,Z 910.061,A -85,B 0,C 180,E1 -5310,E2 -5310} C_VEL
LIN {X 0,Y 509.071,Z 909.79,A -85,B 0,C 180,E1 -5310.791,E2 -5310.791} C_VEL
LIN {X 0,Y 509.112,Z 909.052,A -85,B 0,C 180,E1 -5311.582,E2 -5311.582} C_VEL
LIN {X 0,Y 509.192,Z 907.847,A -85,B 0,C 180,E1 -5312.373,E2 -5312.373} C_VEL
LIN {X 0,Y 509.246,Z 905.005,A -85,B 0,C 180,E1 -5313.561,E2 -5313.561} C_VEL
LIN {X 0,Y 509.312,Z 902.421,A -85,B 0,C 180,E1 -5314.353,E2 -5314.353} C_VEL
LIN {X 0,Y 509.378,Z 897.328,A -85,B 0,C 180,E1 -5315.542,E2 -5315.542} C_VEL
LIN {X 0,Y 509.524,Z 892.227,A -85,B 0,C 180,E1 -5316.469,E2 -5316.469} C_VEL
LIN {X 0,Y 509.651,Z 884.971,A -85,B 0,C 180,E1 -5317.528,E2 -5317.528} C_VEL
LIN {X 0,Y 509.876,Z 876.057,A -85,B 0,C 180,E1 -5318.521,E2 -5318.521} C_VEL
LIN {X 0,Y 510.105,Z 868.308,A -85,B 0,C 180,E1 -5319.216,E2 -5319.216} C_VEL
LIN {X 0,Y 510.256,Z 860.137,A -85,B 0,C 180,E1 -5319.814,E2 -5319.814} C_VEL
LIN {X 0,Y 510.521,Z 849.741,A -85,B 0,C 180,E1 -5320.41,E2 -5320.41} C_VEL
LIN {X 0,Y 510.72,Z 838.024,A -85,B 0,C 180,E1 -5320.882,E2 -5320.882} C_VEL
LIN {X 0,Y 510.897,Z 827.676,A -85,B 0,C 180,E1 -5321.15,E2 -5321.15} C_VEL
LIN {X 0,Y 511.027,Z 760.918,A -85,B 0,C 180,E1 -5322.11,E2 -5322.11} C_VEL
LIN {X 0,Y 509.621,Z 751.769,A -85,B 0,C 180,E1 -5322.297,E2 -5322.297} C_VEL
LIN {X 0,Y 509.927,Z 739.065,A -85,B 0,C 180,E1 -5325.254,E2 -5325.254} C_VEL
LIN {X 0,Y 510.156,Z 727.132,A -85,B 0,C 180,E1 -5328.092,E2 -5328.092} C_VEL
LIN {X 0,Y 509.934,Z 723.854,A -85,B 0,C 180,E1 -5328.95,E2 -5328.95} C_VEL
LIN {X 0,Y 509.823,Z 723.791,A -85,B 0,C 180,E1 -5331.851,E2 -5331.851} C_VEL
LIN {X 0,Y 509.831,Z 723.792,A -85,B 0,C 180,E1 -5334.521,E2 -5334.521} C_VEL
LIN {X 0,Y 509.834,Z 723.786,A -85,B 0,C 180,E1 -5337.059,E2 -5337.059} C_VEL
LIN {X 0,Y 509.858,Z 723.784,A -85,B 0,C 180,E1 -5339.751,E2 -5339.751} C_VEL
LIN {X 0,Y 509.868,Z 723.784,A -85,B 0,C 180,E1 -5342.773,E2 -5342.773} C_VEL
LIN {X 0,Y 509.827,Z 723.787,A -85,B 0,C 180,E1 -5345.578,E2 -5345.578} C_VEL
LIN {X 0,Y 509.85,Z 723.782,A -85,B 0,C 180,E1 -5348.338,E2 -5348.338} C_VEL
LIN {X 0,Y 509.856,Z 723.782,A -85,B 0,C 180,E1 -5351.426,E2 -5351.426} C_VEL
LIN {X 0,Y 509.84,Z 723.787,A -85,B 0,C 180,E1 -5354.67,E2 -5354.67} C_VEL
LIN {X 0,Y 509.855,Z 723.766,A -85,B 0,C 180,E1 -5358.104,E2 -5358.104} C_VEL
LIN {X 0,Y 509.846,Z 723.785,A -85,B 0,C 180,E1 -5360.647,E2 -5360.647} C_VEL
LIN {X 0,Y 509.826,Z 723.786,A -85,B 0,C 180,E1 -5363.647,E2 -5363.647} C_VEL
LIN {X 0,Y 509.843,Z 723.785,A -85,B 0,C 180,E1 -5366.538,E2 -5366.538} C_VEL
LIN {X 0,Y 509.844,Z 723.787,A -85,B 0,C 180,E1 -5369.334,E2 -5369.334} C_VEL
LIN {X 0,Y 509.887,Z 723.777,A -85,B 0,C 180,E1 -5372.054,E2 -5372.054} C_VEL
LIN {X 0,Y 509.876,Z 723.778,A -85,B 0,C 180,E1 -5374.704,E2 -5374.704} C_VEL
LIN {X 0,Y 509.828,Z 723.789,A -85,B 0,C 180,E1 -5377.458,E2 -5377.458} C_VEL
LIN {X 0,Y 509.919,Z 723.774,A -85,B 0,C 180,E1 -5379.845,E2 -5379.845} C_VEL
LIN {X 0,Y 509.877,Z 723.78,A -85,B 0,C 180,E1 -5383.174,E2 -5383.174} C_VEL
LIN {X 0,Y 509.876,Z 723.783,A -85,B 0,C 180,E1 -5385.634,E2 -5385.634} C_VEL
LIN {X 0,Y 509.916,Z 723.778,A -85,B 0,C 180,E1 -5388.874,E2 -5388.874} C_VEL
LIN {X 0,Y 509.953,Z 723.761,A -85,B 0,C 180,E1 -5392.078,E2 -5392.078} C_VEL
LIN {X 0,Y 509.983,Z 723.763,A -85,B 0,C 180,E1 -5394.464,E2 -5394.464} C_VEL
LIN {X 0,Y 510.058,Z 723.763,A -85,B 0,C 180,E1 -5397.631,E2 -5397.631} C_VEL
LIN {X 0,Y 510.066,Z 723.752,A -85,B 0,C 180,E1 -5400.789,E2 -5400.789} C_VEL
LIN {X 0,Y 509.957,Z 723.763,A -85,B 0,C 180,E1 -5403.16,E2 -5403.16} C_VEL
LIN {X 0,Y 509.961,Z 723.77,A -85,B 0,C 180,E1 -5406.33,E2 -5406.33} C_VEL
LIN {X 0,Y 509.918,Z 723.774,A -85,B 0,C 180,E1 -5408.72,E2 -5408.72} C_VEL
LIN {X 0,Y 509.907,Z 723.775,A -85,B 0,C 180,E1 -5411.932,E2 -5411.932} C_VEL
LIN {X 0,Y 509.896,Z 723.777,A -85,B 0,C 180,E1 -5415.242,E2 -5415.242} C_VEL
LIN {X 0,Y 509.891,Z 723.784,A -85,B 0,C 180,E1 -5418.001,E2 -5418.001} C_VEL
LIN {X 0,Y 509.852,Z 723.776,A -85,B 0,C 180,E1 -5421.002,E2 -5421.002} C_VEL
LIN {X 0,Y 509.839,Z 723.785,A -85,B 0,C 180,E1 -5423.563,E2 -5423.563} C_VEL
LIN {X 0,Y 509.914,Z 723.779,A -85,B 0,C 180,E1 -5426.379,E2 -5426.379} C_VEL
LIN {X 0,Y 509.879,Z 723.774,A -85,B 0,C 180,E1 -5428.844,E2 -5428.844} C_VEL
LIN {X 0,Y 509.823,Z 723.786,A -85,B 0,C 180,E1 -5431.59,E2 -5431.59} C_VEL
LIN {X 0,Y 509.856,Z 723.786,A -85,B 0,C 180,E1 -5434.413,E2 -5434.413} C_VEL
LIN {X 0,Y 509.821,Z 723.778,A -85,B 0,C 180,E1 -5437.34,E2 -5437.34} C_VEL
LIN {X 0,Y 509.863,Z 723.773,A -85,B 0,C 180,E1 -5440.38,E2 -5440.38} C_VEL
LIN {X 0,Y 509.825,Z 723.786,A -85,B 0,C 180,E1 -5443.062,E2 -5443.062} C_VEL
LIN {X 0,Y 509.831,Z 723.787,A -85,B 0,C 180,E1 -5445.792,E2 -5445.792} C_VEL
LIN {X 0,Y 509.86,Z 723.782,A -85,B 0,C 180,E1 -5448.575,E2 -5448.575} C_VEL
LIN {X 0,Y 509.853,Z 723.784,A -85,B 0,C 180,E1 -5451.786,E2 -5451.786} C_VEL
LIN {X 0,Y 509.848,Z 723.788,A -85,B 0,C 180,E1 -5454.623,E2 -5454.623} C_VEL
LIN {X 0,Y 509.867,Z 723.78,A -85,B 0,C 180,E1 -5457.481,E2 -5457.481} C_VEL
LIN {X 0,Y 509.859,Z 723.779,A -85,B 0,C 180,E1 -5460.274,E2 -5460.274} C_VEL
LIN {X 0,Y 509.886,Z 723.78,A -85,B 0,C 180,E1 -5462.944,E2 -5462.944} C_VEL
LIN {X 0,Y 509.857,Z 723.782,A -85,B 0,C 180,E1 -5465.573,E2 -5465.573} C_VEL
LIN {X 0,Y 509.891,Z 723.916,A -85,B 0,C 180,E1 -5467.138,E2 -5467.138} C_VEL
LIN {X 0,Y 510.885,Z 730.091,A -85,B 0,C 180,E1 -5468.408,E2 -5468.408} C_VEL
LIN {X 0,Y 510.549,Z 745.392,A -85,B 0,C 180,E1 -5471.334,E2 -5471.334} C_VEL
LIN {X 0,Y 510.157,Z 761.692,A -85,B 0,C 180,E1 -5474.402,E2 -5474.402} C_VEL
LIN {X 0,Y 509.825,Z 777.034,A -85,B 0,C 180,E1 -5477.258,E2 -5477.258} C_VEL
LIN {X 0,Y 509.795,Z 779.828,A -85,B 0,C 180,E1 -5477.728,E2 -5477.728} C_VEL
LIN {X 0,Y 510.523,Z 785.506,A -85,B 0,C 180,E1 -5477.855,E2 -5477.855} C_VEL
LIN {X 0,Y 511.073,Z 791.864,A -85,B 0,C 180,E1 -5477.957,E2 -5477.957} C_VEL
LIN {X 0,Y 510.88,Z 855.988,A -85,B 0,C 180,E1 -5478.872,E2 -5478.872} C_VEL
LIN {X 0,Y 510.702,Z 865.198,A -85,B 0,C 180,E1 -5479.093,E2 -5479.093} C_VEL
LIN {X 0,Y 510.609,Z 873.683,A -85,B 0,C 180,E1 -5479.392,E2 -5479.392} C_VEL
LIN {X 0,Y 510.435,Z 882.203,A -85,B 0,C 180,E1 -5479.789,E2 -5479.789} C_VEL
LIN {X 0,Y 510.222,Z 890.554,A -85,B 0,C 180,E1 -5480.286,E2 -5480.286} C_VEL
LIN {X 0,Y 510.043,Z 898.613,A -85,B 0,C 180,E1 -5480.882,E2 -5480.882} C_VEL
LIN {X 0,Y 509.794,Z 907.311,A -85,B 0,C 180,E1 -5481.677,E2 -5481.677} C_VEL
LIN {X 0,Y 509.621,Z 915.849,A -85,B 0,C 180,E1 -5482.671,E2 -5482.671} C_VEL
LIN {X 0,Y 509.484,Z 922.549,A -85,B 0,C 180,E1 -5483.664,E2 -5483.664} C_VEL
LIN {X 0,Y 509.382,Z 926.947,A -85,B 0,C 180,E1 -5484.458,E2 -5484.458} C_VEL
LIN {X 0,Y 509.297,Z 932.133,A -85,B 0,C 180,E1 -5485.647,E2 -5485.647} C_VEL
LIN {X 0,Y 509.247,Z 934.782,A -85,B 0,C 180,E1 -5486.439,E2 -5486.439} C_VEL
LIN {X 0,Y 509.161,Z 937.68,A -85,B 0,C 180,E1 -5487.627,E2 -5487.627} C_VEL
LIN {X 0,Y 509.111,Z 938.928,A -85,B 0,C 180,E1 -5488.418,E2 -5488.418} C_VEL
LIN {X 0,Y 509.071,Z 939.706,A -85,B 0,C 180,E1 -5489.209,E2 -5489.209} C_VEL
LIN {X 0,Y 509.062,Z 940,A -85,B 0,C 180,E1 -5490,E2 -5490} C_VEL
LIN {X 0,Y 509.071,Z 939.705,A -85,B 0,C 180,E1 -5490.791,E2 -5490.791} C_VEL
LIN {X 0,Y 509.111,Z 938.927,A -85,B 0,C 180,E1 -5491.582,E2 -5491.582} C_VEL
LIN {X 0,Y 509.161,Z 937.679,A -85,B 0,C 180,E1 -5492.373,E2 -5492.373} C_VEL
LIN {X 0,Y 509.247,Z 934.781,A -85,B 0,C 180,E1 -5493.561,E2 -5493.561} C_VEL
LIN {X 0,Y 509.297,Z 932.132,A -85,B 0,C 180,E1 -5494.353,E2 -5494.353} C_VEL
LIN {X 0,Y 509.382,Z 926.944,A -85,B 0,C 180,E1 -5495.542,E2 -5495.542} C_VEL
LIN {X 0,Y 509.49,Z 921.79,A -85,B 0,C 180,E1 -5496.463,E2 -5496.463} C_VEL
LIN {X 0,Y 509.624,Z 914.339,A -85,B 0,C 180,E1 -5497.528,E2 -5497.528} C_VEL
LIN {X 0,Y 509.829,Z 906.295,A -85,B 0,C 180,E1 -5498.422,E2 -5498.422} C_VEL
LIN {X 0,Y 510.043,Z 898.617,A -85,B 0,C 180,E1 -5499.118,E2 -5499.118} C_VEL
LIN {X 0,Y 510.222,Z 890.555,A -85,B 0,C 180,E1 -5499.714,E2 -5499.714} C_VEL
LIN {X 0,Y 510.435,Z 882.205,A -85,B 0,C 180,E1 -5500.211,E2 -5500.211} C_VEL
LIN {X 0,Y 510.619,Z 873.687,A -85,B 0,C 180,E1 -5500.608,E2 -5500.608} C_VEL
LIN {X 0,Y 510.753,Z 863.537,A -85,B 0,C 180,E1 -5500.956,E2 -5500.956} C_VEL
LIN {X 0,Y 510.951,Z 852.239,A -85,B 0,C 180,E1 -5501.197,E2 -5501.197} C_VEL
LIN {X 0,Y 510.909,Z 788.471,A -85,B 0,C 180,E1 -5502.094,E2 -5502.094} C_VEL
LIN {X 0,Y 509.785,Z 779.866,A -85,B 0,C 180,E1 -5502.268,E2 -5502.268} C_VEL
LIN {X 0,Y 509.887,Z 773.758,A -85,B 0,C 180,E1 -5503.348,E2 -5503.348} C_VEL
LIN {X 0,Y 510.241,Z 758.474,A -85,B 0,C 180,E1 -5506.196,E2 -5506.196} C_VEL
LIN {X 0,Y 510.641,Z 741.019,A -85,B 0,C 180,E1 -5509.497,E2 -5509.497} C_VEL
LIN {X 0,Y 510.891,Z 730.091,A -85,B 0,C 180,E1 -5511.591,E2 -5511.591} C_VEL
LIN {X 0,Y 509.864,Z 723.861,A -85,B 0,C 180,E1 -5512.89,E2 -5512.89} C_VEL
LIN {X 0,Y 509.91,Z 723.775,A -85,B 0,C 180,E1 -5516.171,E2 -5516.171} C_VEL
LIN {X 0,Y 509.878,Z 723.785,A -85,B 0,C 180,E1 -5518.844,E2 -5518.844} C_VEL
LIN {X 0,Y 509.827,Z 723.789,A -85,B 0,C 180,E1 -5521.59,E2 -5521.59} C_VEL
LIN {X 0,Y 509.855,Z 723.783,A -85,B 0,C 180,E1 -5524.413,E2 -5524.413} C_VEL
LIN {X 0,Y 509.82,Z 723.793,A -85,B 0,C 180,E1 -5527.341,E2 -5527.341} C_VEL
LIN {X 0,Y 509.84,Z 723.78,A -85,B 0,C 180,E1 -5530.382,E2 -5530.382} C_VEL
LIN {X 0,Y 509.825,Z 723.785,A -85,B 0,C 180,E1 -5533.062,E2 -5533.062} C_VEL
LIN {X 0,Y 509.832,Z 723.791,A -85,B 0,C 180,E1 -5535.792,E2 -5535.792} C_VEL
LIN {X 0,Y 509.867,Z 723.773,A -85,B 0,C 180,E1 -5538.576,E2 -5538.576} C_VEL
LIN {X 0,Y 509.854,Z 723.774,A -85,B 0,C 180,E1 -5541.786,E2 -5541.786} C_VEL
LIN {X 0,Y 509.848,Z 723.782,A -85,B 0,C 180,E1 -5544.623,E2 -5544.623} C_VEL
LIN {X 0,Y 509.865,Z 723.785,A -85,B 0,C 180,E1 -5547.481,E2 -5547.481} C_VEL
LIN {X 0,Y 509.86,Z 723.78,A -85,B 0,C 180,E1 -5550.274,E2 -5550.274} C_VEL
LIN {X 0,Y 509.887,Z 723.778,A -85,B 0,C 180,E1 -5552.945,E2 -5552.945} C_VEL
LIN {X 0,Y 509.872,Z 723.783,A -85,B 0,C 180,E1 -5555.574,E2 -5555.574} C_VEL
LIN {X 0,Y 509.825,Z 723.787,A -85,B 0,C 180,E1 -5558.149,E2 -5558.149} C_VEL
LIN {X 0,Y 509.867,Z 723.781,A -85,B 0,C 180,E1 -5560.682,E2 -5560.682} C_VEL
LIN {X 0,Y 509.889,Z 723.778,A -85,B 0,C 180,E1 -5563.175,E2 -5563.175} C_VEL
LIN {X 0,Y 509.866,Z 723.78,A -85,B 0,C 180,E1 -5565.634,E2 -5565.634} C_VEL
LIN {X 0,Y 509.915,Z 723.772,A -85,B 0,C 180,E1 -5568.875,E2 -5568.875} C_VEL
LIN {X 0,Y 509.954,Z 723.775,A -85,B 0,C 180,E1 -5572.079,E2 -5572.079} C_VEL
LIN {X 0,Y 509.983,Z 723.772,A -85,B 0,C 180,E1 -5574.464,E2 -5574.464} C_VEL
LIN {X 0,Y 510.058,Z 723.748,A -85,B 0,C 180,E1 -5577.631,E2 -5577.631} C_VEL
LIN {X 0,Y 510.066,Z 723.761,A -85,B 0,C 180,E1 -5580.79,E2 -5580.79} C_VEL
LIN {X 0,Y 509.958,Z 723.771,A -85,B 0,C 180,E1 -5583.16,E2 -5583.16} C_VEL
LIN {X 0,Y 509.956,Z 723.771,A -85,B 0,C 180,E1 -5586.33,E2 -5586.33} C_VEL
LIN {X 0,Y 509.914,Z 723.776,A -85,B 0,C 180,E1 -5588.72,E2 -5588.72} C_VEL
LIN {X 0,Y 509.907,Z 723.776,A -85,B 0,C 180,E1 -5591.932,E2 -5591.932} C_VEL
LIN {X 0,Y 509.896,Z 723.776,A -85,B 0,C 180,E1 -5595.242,E2 -5595.242} C_VEL
LIN {X 0,Y 509.869,Z 723.774,A -85,B 0,C 180,E1 -5597.993,E2 -5597.993} C_VEL
LIN {X 0,Y 509.888,Z 723.779,A -85,B 0,C 180,E1 -5600.402,E2 -5600.402} C_VEL
LIN {X 0,Y 509.824,Z 723.786,A -85,B 0,C 180,E1 -5603.564,E2 -5603.564} C_VEL
LIN {X 0,Y 509.912,Z 723.769,A -85,B 0,C 180,E1 -5606.378,E2 -5606.378} C_VEL
LIN {X 0,Y 509.876,Z 723.784,A -85,B 0,C 180,E1 -5608.844,E2 -5608.844} C_VEL
LIN {X 0,Y 509.82,Z 723.787,A -85,B 0,C 180,E1 -5611.59,E2 -5611.59} C_VEL
LIN {X 0,Y 509.84,Z 723.781,A -85,B 0,C 180,E1 -5614.414,E2 -5614.414} C_VEL
LIN {X 0,Y 509.817,Z 723.795,A -85,B 0,C 180,E1 -5617.341,E2 -5617.341} C_VEL
LIN {X 0,Y 509.839,Z 723.778,A -85,B 0,C 180,E1 -5620.382,E2 -5620.382} C_VEL
LIN {X 0,Y 509.808,Z 723.774,A -85,B 0,C 180,E1 -5623.06,E2 -5623.06} C_VEL
LIN {X 0,Y 509.824,Z 723.79,A -85,B 0,C 180,E1 -5625.793,E2 -5625.793} C_VEL
LIN {X 0,Y 509.856,Z 723.782,A -85,B 0,C 180,E1 -5628.574,E2 -5628.574} C_VEL
LIN {X 0,Y 509.852,Z 723.782,A -85,B 0,C 180,E1 -5631.787,E2 -5631.787} C_VEL
LIN {X 0,Y 509.822,Z 723.792,A -85,B 0,C 180,E1 -5633.733,E2 -5633.733} C_VEL
LIN {X 0,Y 509.153,Z 723.873,A -85,B 0,C 180,E1 -5634.392,E2 -5634.392} C_VEL
LIN {X 0,Y 506.34,Z 724.228,A -85,B 0,C 180,E1 -5635.464,E2 -5635.464} C_VEL
LIN {X 0,Y 503.953,Z 724.523,A -85,B 0,C 180,E1 -5636.328,E2 -5636.328} C_VEL
LIN {X 0,Y 502.906,Z 724.649,A -85,B 0,C 180,E1 -5636.994,E2 -5636.994} C_VEL
LIN {X 0,Y 502.808,Z 724.66,A -85,B 0,C 180,E1 -5637.22,E2 -5637.22} C_VEL
LIN {X 0,Y 502.816,Z 724.665,A -85,B 0,C 180,E1 -5640.065,E2 -5640.065} C_VEL
LIN {X 0,Y 502.845,Z 724.661,A -85,B 0,C 180,E1 -5643.444,E2 -5643.444} C_VEL
LIN {X 0,Y 502.789,Z 724.662,A -85,B 0,C 180,E1 -5646.959,E2 -5646.959} C_VEL
LIN {X 0,Y 502.845,Z 724.663,A -85,B 0,C 180,E1 -5650.401,E2 -5650.401} C_VEL
LIN {X 0,Y 502.952,Z 724.921,A -85,B 0,C 180,E1 -5651.147,E2 -5651.147} C_VEL
LIN {X 0,Y 503.153,Z 730.516,A -85,B 0,C 180,E1 -5652.524,E2 -5652.524} C_VEL
LIN {X 0,Y 502.819,Z 742.629,A -85,B 0,C 180,E1 -5655.428,E2 -5655.428} C_VEL
LIN {X 0,Y 502.608,Z 751.99,A -85,B 0,C 180,E1 -5657.596,E2 -5657.596} C_VEL
LIN {X 0,Y 503.032,Z 754.567,A -85,B 0,C 180,E1 -5657.691,E2 -5657.691} C_VEL
LIN {X 0,Y 504.153,Z 762.855,A -85,B 0,C 180,E1 -5657.837,E2 -5657.837} C_VEL
LIN {X 0,Y 503.892,Z 826.941,A -85,B 0,C 180,E1 -5658.765,E2 -5658.765} C_VEL
LIN {X 0,Y 503.785,Z 836.098,A -85,B 0,C 180,E1 -5658.992,E2 -5658.992} C_VEL
LIN {X 0,Y 503.67,Z 844.506,A -85,B 0,C 180,E1 -5659.295,E2 -5659.295} C_VEL
LIN {X 0,Y 503.495,Z 852.027,A -85,B 0,C 180,E1 -5659.647,E2 -5659.647} C_VEL
LIN {X 0,Y 503.273,Z 860.508,A -85,B 0,C 180,E1 -5660.15,E2 -5660.15} C_VEL
LIN {X 0,Y 503.136,Z 868.646,A -85,B 0,C 180,E1 -5660.756,E2 -5660.756} C_VEL
LIN {X 0,Y 502.843,Z 876.374,A -85,B 0,C 180,E1 -5661.46,E2 -5661.46} C_VEL
LIN {X 0,Y 502.61,Z 884.448,A -85,B 0,C 180,E1 -5662.366,E2 -5662.366} C_VEL
LIN {X 0,Y 502.487,Z 891.717,A -85,B 0,C 180,E1 -5663.407,E2 -5663.407} C_VEL
LIN {X 0,Y 502.337,Z 897.106,A -85,B 0,C 180,E1 -5664.38,E2 -5664.38} C_VEL
LIN {X 0,Y 502.154,Z 900.782,A -85,B 0,C 180,E1 -5665.183,E2 -5665.183} C_VEL
LIN {X 0,Y 502.252,Z 903.774,A -85,B 0,C 180,E1 -5665.988,E2 -5665.988} C_VEL
LIN {X 0,Y 502.135,Z 906.102,A -85,B 0,C 180,E1 -5666.791,E2 -5666.791} C_VEL
LIN {X 0,Y 502.123,Z 907.873,A -85,B 0,C 180,E1 -5667.593,E2 -5667.593} C_VEL
LIN {X 0,Y 502.035,Z 909.152,A -85,B 0,C 180,E1 -5668.396,E2 -5668.396} C_VEL
LIN {X 0,Y 501.987,Z 909.962,A -85,B 0,C 180,E1 -5669.198,E2 -5669.198} C_VEL
LIN {X 0,Y 501.978,Z 910.269,A -85,B 0,C 180,E1 -5670,E2 -5670} C_VEL
LIN {X 0,Y 501.988,Z 909.998,A -85,B 0,C 180,E1 -5670.802,E2 -5670.802} C_VEL
LIN {X 0,Y 502.036,Z 909.259,A -85,B 0,C 180,E1 -5671.604,E2 -5671.604} C_VEL
LIN {X 0,Y 502.123,Z 908.054,A -85,B 0,C 180,E1 -5672.407,E2 -5672.407} C_VEL
LIN {X 0,Y 502.172,Z 905.212,A -85,B 0,C 180,E1 -5673.611,E2 -5673.611} C_VEL
LIN {X 0,Y 502.236,Z 902.627,A -85,B 0,C 180,E1 -5674.414,E2 -5674.414} C_VEL
LIN {X 0,Y 502.328,Z 897.533,A -85,B 0,C 180,E1 -5675.62,E2 -5675.62} C_VEL
LIN {X 0,Y 502.451,Z 893.22,A -85,B 0,C 180,E1 -5676.425,E2 -5676.425} C_VEL
LIN {X 0,Y 502.521,Z 888.044,A -85,B 0,C 180,E1 -5677.231,E2 -5677.231} C_VEL
LIN {X 0,Y 502.683,Z 881.808,A -85,B 0,C 180,E1 -5678.037,E2 -5678.037} C_VEL
LIN {X 0,Y 502.95,Z 874.219,A -85,B 0,C 180,E1 -5678.842,E2 -5678.842} C_VEL
LIN {X 0,Y 503.193,Z 864.779,A -85,B 0,C 180,E1 -5679.648,E2 -5679.648} C_VEL
LIN {X 0,Y 503.42,Z 855.551,A -85,B 0,C 180,E1 -5680.253,E2 -5680.253} C_VEL
LIN {X 0,Y 503.61,Z 846.642,A -85,B 0,C 180,E1 -5680.707,E2 -5680.707} C_VEL
LIN {X 0,Y 503.784,Z 837.372,A -85,B 0,C 180,E1 -5681.059,E2 -5681.059} C_VEL
LIN {X 0,Y 503.951,Z 827.956,A -85,B 0,C 180,E1 -5681.303,E2 -5681.303} C_VEL
LIN {X 0,Y 504.078,Z 761.463,A -85,B 0,C 180,E1 -5682.274,E2 -5682.274} C_VEL
LIN {X 0,Y 502.59,Z 751.865,A -85,B 0,C 180,E1 -5682.472,E2 -5682.472} C_VEL
LIN {X 0,Y 502.909,Z 739.541,A -85,B 0,C 180,E1 -5685.398,E2 -5685.398} C_VEL
LIN {X 0,Y 503.159,Z 727.789,A -85,B 0,C 180,E1 -5688.23,E2 -5688.23} C_VEL
LIN {X 0,Y 502.881,Z 724.753,A -85,B 0,C 180,E1 -5689.014,E2 -5689.014} C_VEL
LIN {X 0,Y 502.781,Z 724.673,A -85,B 0,C 180,E1 -5692.174,E2 -5692.174} C_VEL
LIN {X 0,Y 502.771,Z 724.669,A -85,B 0,C 180,E1 -5694.794,E2 -5694.794} C_VEL
LIN {X 0,Y 502.789,Z 724.664,A -85,B 0,C 180,E1 -5697.469,E2 -5697.469} C_VEL
LIN {X 0,Y 502.809,Z 724.668,A -85,B 0,C 180,E1 -5700.211,E2 -5700.211} C_VEL
LIN {X 0,Y 502.83,Z 724.659,A -85,B 0,C 180,E1 -5703.031,E2 -5703.031} C_VEL
LIN {X 0,Y 502.775,Z 724.668,A -85,B 0,C 180,E1 -5705.951,E2 -5705.951} C_VEL
LIN {X 0,Y 502.798,Z 724.659,A -85,B 0,C 180,E1 -5708.976,E2 -5708.976} C_VEL
LIN {X 0,Y 502.796,Z 724.665,A -85,B 0,C 180,E1 -5712.139,E2 -5712.139} C_VEL
LIN {X 0,Y 502.787,Z 724.656,A -85,B 0,C 180,E1 -5715.47,E2 -5715.47} C_VEL
LIN {X 0,Y 502.821,Z 724.655,A -85,B 0,C 180,E1 -5718.934,E2 -5718.934} C_VEL
LIN {X 0,Y 502.794,Z 724.662,A -85,B 0,C 180,E1 -5722.046,E2 -5722.046} C_VEL
LIN {X 0,Y 502.797,Z 724.664,A -85,B 0,C 180,E1 -5725.034,E2 -5725.034} C_VEL
LIN {X 0,Y 502.784,Z 724.66,A -85,B 0,C 180,E1 -5727.915,E2 -5727.915} C_VEL
LIN {X 0,Y 502.824,Z 724.664,A -85,B 0,C 180,E1 -5730.712,E2 -5730.712} C_VEL
LIN {X 0,Y 502.865,Z 724.649,A -85,B 0,C 180,E1 -5733.439,E2 -5733.439} C_VEL
LIN {X 0,Y 502.786,Z 724.66,A -85,B 0,C 180,E1 -5736.086,E2 -5736.086} C_VEL
LIN {X 0,Y 502.785,Z 724.666,A -85,B 0,C 180,E1 -5738.689,E2 -5738.689} C_VEL
LIN {X 0,Y 502.829,Z 724.659,A -85,B 0,C 180,E1 -5741.248,E2 -5741.248} C_VEL
LIN {X 0,Y 502.851,Z 724.651,A -85,B 0,C 180,E1 -5744.6,E2 -5744.6} C_VEL
LIN {X 0,Y 502.879,Z 724.652,A -85,B 0,C 180,E1 -5748.039,E2 -5748.039} C_VEL
LIN {X 0,Y 502.872,Z 724.655,A -85,B 0,C 180,E1 -5751.157,E2 -5751.157} C_VEL
LIN {X 0,Y 502.909,Z 724.65,A -85,B 0,C 180,E1 -5753.581,E2 -5753.581} C_VEL
LIN {X 0,Y 502.901,Z 724.649,A -85,B 0,C 180,E1 -5756.795,E2 -5756.795} C_VEL
LIN {X 0,Y 503.036,Z 724.636,A -85,B 0,C 180,E1 -5759.199,E2 -5759.199} C_VEL
LIN {X 0,Y 502.903,Z 724.646,A -85,B 0,C 180,E1 -5761.602,E2 -5761.602} C_VEL
LIN {X 0,Y 502.9,Z 724.642,A -85,B 0,C 180,E1 -5763.204,E2 -5763.204} C_VEL
LIN {X 0,Y 502.913,Z 724.647,A -85,B 0,C 180,E1 -5766.419,E2 -5766.419} C_VEL
LIN {X 0,Y 502.876,Z 724.651,A -85,B 0,C 180,E1 -5768.843,E2 -5768.843} C_VEL
LIN {X 0,Y 502.848,Z 724.652,A -85,B 0,C 180,E1 -5772.102,E2 -5772.102} C_VEL
LIN {X 0,Y 502.851,Z 724.656,A -85,B 0,C 180,E1 -5775.4,E2 -5775.4} C_VEL
LIN {X 0,Y 502.849,Z 724.659,A -85,B 0,C 180,E1 -5778.122,E2 -5778.122} C_VEL
LIN {X 0,Y 502.83,Z 724.651,A -85,B 0,C 180,E1 -5780.536,E2 -5780.536} C_VEL
LIN {X 0,Y 502.799,Z 724.658,A -85,B 0,C 180,E1 -5783.04,E2 -5783.04} C_VEL
LIN {X 0,Y 502.842,Z 724.66,A -85,B 0,C 180,E1 -5785.675,E2 -5785.675} C_VEL
LIN {X 0,Y 502.842,Z 724.655,A -85,B 0,C 180,E1 -5788.372,E2 -5788.372} C_VEL
LIN {X 0,Y 502.795,Z 724.661,A -85,B 0,C 180,E1 -5791.499,E2 -5791.499} C_VEL
LIN {X 0,Y 502.808,Z 724.664,A -85,B 0,C 180,E1 -5794.445,E2 -5794.445} C_VEL
LIN {X 0,Y 502.783,Z 724.654,A -85,B 0,C 180,E1 -5797.178,E2 -5797.178} C_VEL
LIN {X 0,Y 502.823,Z 724.642,A -85,B 0,C 180,E1 -5800.012,E2 -5800.012} C_VEL
LIN {X 0,Y 502.774,Z 724.663,A -85,B 0,C 180,E1 -5803.231,E2 -5803.231} C_VEL
LIN {X 0,Y 502.79,Z 724.663,A -85,B 0,C 180,E1 -5805.661,E2 -5805.661} C_VEL
LIN {X 0,Y 502.82,Z 724.657,A -85,B 0,C 180,E1 -5809.005,E2 -5809.005} C_VEL
LIN {X 0,Y 502.796,Z 724.665,A -85,B 0,C 180,E1 -5812.046,E2 -5812.046} C_VEL
LIN {X 0,Y 502.811,Z 724.664,A -85,B 0,C 180,E1 -5815.035,E2 -5815.035} C_VEL
LIN {X 0,Y 502.789,Z 724.661,A -85,B 0,C 180,E1 -5817.916,E2 -5817.916} C_VEL
LIN {X 0,Y 502.825,Z 724.661,A -85,B 0,C 180,E1 -5820.712,E2 -5820.712} C_VEL
LIN {X 0,Y 502.863,Z 724.653,A -85,B 0,C 180,E1 -5823.439,E2 -5823.439} C_VEL
LIN {X 0,Y 502.811,Z 724.664,A -85,B 0,C 180,E1 -5826.525,E2 -5826.525} C_VEL
LIN {X 0,Y 502.825,Z 724.698,A -85,B 0,C 180,E1 -5826.961,E2 -5826.961} C_VEL
LIN {X 0,Y 503.901,Z 731.013,A -85,B 0,C 180,E1 -5828.309,E2 -5828.309} C_VEL
LIN {X 0,Y 503.545,Z 746.311,A -85,B 0,C 180,E1 -5831.276,E2 -5831.276} C_VEL
LIN {X 0,Y 503.108,Z 761.812,A -85,B 0,C 180,E1 -5834.234,E2 -5834.234} C_VEL
LIN {X 0,Y 502.803,Z 775.753,A -85,B 0,C 180,E1 -5836.871,E2 -5836.871} C_VEL
LIN {X 0,Y 502.756,Z 779.68,A -85,B 0,C 180,E1 -5837.558,E2 -5837.558} C_VEL
LIN {X 0,Y 504.131,Z 791.656,A -85,B 0,C 180,E1 -5837.789,E2 -5837.789} C_VEL
LIN {X 0,Y 503.894,Z 857.009,A -85,B 0,C 180,E1 -5838.74,E2 -5838.74} C_VEL
LIN {X 0,Y 503.734,Z 866.654,A -85,B 0,C 180,E1 -5838.991,E2 -5838.991} C_VEL
LIN {X 0,Y 503.492,Z 878.205,A -85,B 0,C 180,E1 -5839.443,E2 -5839.443} C_VEL
LIN {X 0,Y 503.275,Z 888.842,A -85,B 0,C 180,E1 -5840.049,E2 -5840.049} C_VEL
LIN {X 0,Y 503.057,Z 897.172,A -85,B 0,C 180,E1 -5840.653,E2 -5840.653} C_VEL
LIN {X 0,Y 502.798,Z 905.054,A -85,B 0,C 180,E1 -5841.358,E2 -5841.358} C_VEL
LIN {X 0,Y 502.607,Z 912.426,A -85,B 0,C 180,E1 -5842.164,E2 -5842.164} C_VEL
LIN {X 0,Y 502.463,Z 918.918,A -85,B 0,C 180,E1 -5843.031,E2 -5843.031} C_VEL
LIN {X 0,Y 502.362,Z 925.777,A -85,B 0,C 180,E1 -5844.179,E2 -5844.179} C_VEL
LIN {X 0,Y 502.15,Z 930.396,A -85,B 0,C 180,E1 -5845.183,E2 -5845.183} C_VEL
LIN {X 0,Y 502.198,Z 933.403,A -85,B 0,C 180,E1 -5845.988,E2 -5845.988} C_VEL
LIN {X 0,Y 502.134,Z 935.731,A -85,B 0,C 180,E1 -5846.791,E2 -5846.791} C_VEL
LIN {X 0,Y 502.066,Z 937.481,A -85,B 0,C 180,E1 -5847.593,E2 -5847.593} C_VEL
LIN {X 0,Y 502.034,Z 938.736,A -85,B 0,C 180,E1 -5848.396,E2 -5848.396} C_VEL
LIN {X 0,Y 501.988,Z 939.517,A -85,B 0,C 180,E1 -5849.198,E2 -5849.198} C_VEL
LIN {X 0,Y 501.977,Z 939.812,A -85,B 0,C 180,E1 -5850,E2 -5850} C_VEL
LIN {X 0,Y 501.988,Z 939.516,A -85,B 0,C 180,E1 -5850.802,E2 -5850.802} C_VEL
LIN {X 0,Y 502.034,Z 938.735,A -85,B 0,C 180,E1 -5851.604,E2 -5851.604} C_VEL
LIN {X 0,Y 502.066,Z 937.48,A -85,B 0,C 180,E1 -5852.407,E2 -5852.407} C_VEL
LIN {X 0,Y 502.171,Z 934.574,A -85,B 0,C 180,E1 -5853.611,E2 -5853.611} C_VEL
LIN {X 0,Y 502.185,Z 931.922,A -85,B 0,C 180,E1 -5854.415,E2 -5854.415} C_VEL
LIN {X 0,Y 502.308,Z 926.735,A -85,B 0,C 180,E1 -5855.621,E2 -5855.621} C_VEL
LIN {X 0,Y 502.42,Z 920.717,A -85,B 0,C 180,E1 -5856.701,E2 -5856.701} C_VEL
LIN {X 0,Y 502.558,Z 914.13,A -85,B 0,C 180,E1 -5857.634,E2 -5857.634} C_VEL
LIN {X 0,Y 502.777,Z 906.085,A -85,B 0,C 180,E1 -5858.541,E2 -5858.541} C_VEL
LIN {X 0,Y 503.01,Z 898.408,A -85,B 0,C 180,E1 -5859.246,E2 -5859.246} C_VEL
LIN {X 0,Y 503.207,Z 890.346,A -85,B 0,C 180,E1 -5859.851,E2 -5859.851} C_VEL
LIN {X 0,Y 503.434,Z 881.996,A -85,B 0,C 180,E1 -5860.354,E2 -5860.354} C_VEL
LIN {X 0,Y 503.655,Z 873.479,A -85,B 0,C 180,E1 -5860.756,E2 -5860.756} C_VEL
LIN {X 0,Y 503.756,Z 863.327,A -85,B 0,C 180,E1 -5861.11,E2 -5861.11} C_VEL
LIN {X 0,Y 504.009,Z 850.772,A -85,B 0,C 180,E1 -5861.372,E2 -5861.372} C_VEL
LIN {X 0,Y 504.054,Z 789.682,A -85,B 0,C 180,E1 -5862.241,E2 -5862.241} C_VEL
LIN {X 0,Y 502.752,Z 779.654,A -85,B 0,C 180,E1 -5862.442,E2 -5862.442} C_VEL
LIN {X 0,Y 503.035,Z 765.936,A -85,B 0,C 180,E1 -5864.979,E2 -5864.979} C_VEL
LIN {X 0,Y 503.341,Z 751.758,A -85,B 0,C 180,E1 -5867.679,E2 -5867.679} C_VEL
LIN {X 0,Y 503.785,Z 737.571,A -85,B 0,C 180,E1 -5870.412,E2 -5870.412} C_VEL
LIN {X 0,Y 503.896,Z 731.017,A -85,B 0,C 180,E1 -5871.691,E2 -5871.691} C_VEL
LIN {X 0,Y 502.825,Z 724.699,A -85,B 0,C 180,E1 -5873.039,E2 -5873.039} C_VEL
LIN {X 0,Y 502.839,Z 724.659,A -85,B 0,C 180,E1 -5875.676,E2 -5875.676} C_VEL
LIN {X 0,Y 502.841,Z 724.659,A -85,B 0,C 180,E1 -5878.373,E2 -5878.373} C_VEL
LIN {X 0,Y 502.798,Z 724.663,A -85,B 0,C 180,E1 -5881.5,E2 -5881.5} C_VEL
LIN {X 0,Y 502.808,Z 724.661,A -85,B 0,C 180,E1 -5884.445,E2 -5884.445} C_VEL
LIN {X 0,Y 502.782,Z 724.667,A -85,B 0,C 180,E1 -5887.178,E2 -5887.178} C_VEL
LIN {X 0,Y 502.79,Z 724.66,A -85,B 0,C 180,E1 -5890.015,E2 -5890.015} C_VEL
LIN {X 0,Y 502.803,Z 724.658,A -85,B 0,C 180,E1 -5892.199,E2 -5892.199} C_VEL
LIN {X 0,Y 502.802,Z 724.668,A -85,B 0,C 180,E1 -5895.468,E2 -5895.468} C_VEL
LIN {X 0,Y 502.828,Z 724.65,A -85,B 0,C 180,E1 -5899.004,E2 -5899.004} C_VEL
LIN {X 0,Y 502.796,Z 724.658,A -85,B 0,C 180,E1 -5902.046,E2 -5902.046} C_VEL
LIN {X 0,Y 502.811,Z 724.658,A -85,B 0,C 180,E1 -5905.035,E2 -5905.035} C_VEL
LIN {X 0,Y 502.786,Z 724.67,A -85,B 0,C 180,E1 -5907.916,E2 -5907.916} C_VEL
LIN {X 0,Y 502.826,Z 724.653,A -85,B 0,C 180,E1 -5910.712,E2 -5910.712} C_VEL
LIN {X 0,Y 502.864,Z 724.655,A -85,B 0,C 180,E1 -5913.439,E2 -5913.439} C_VEL
LIN {X 0,Y 502.794,Z 724.667,A -85,B 0,C 180,E1 -5916.086,E2 -5916.086} C_VEL
LIN {X 0,Y 502.786,Z 724.657,A -85,B 0,C 180,E1 -5918.689,E2 -5918.689} C_VEL
LIN {X 0,Y 502.833,Z 724.656,A -85,B 0,C 180,E1 -5921.248,E2 -5921.248} C_VEL
LIN {X 0,Y 502.826,Z 724.661,A -85,B 0,C 180,E1 -5923.767,E2 -5923.767} C_VEL
LIN {X 0,Y 502.833,Z 724.658,A -85,B 0,C 180,E1 -5926.255,E2 -5926.255} C_VEL
LIN {X 0,Y 502.879,Z 724.65,A -85,B 0,C 180,E1 -5928.717,E2 -5928.717} C_VEL
LIN {X 0,Y 502.904,Z 724.651,A -85,B 0,C 180,E1 -5931.967,E2 -5931.967} C_VEL
LIN {X 0,Y 502.937,Z 724.651,A -85,B 0,C 180,E1 -5934.387,E2 -5934.387} C_VEL
LIN {X 0,Y 503.027,Z 724.623,A -85,B 0,C 180,E1 -5937.598,E2 -5937.598} C_VEL
LIN {X 0,Y 503.03,Z 724.63,A -85,B 0,C 180,E1 -5940,E2 -5940} C_VEL
LIN {X 0,Y 503.028,Z 724.639,A -85,B 0,C 180,E1 -5942.402,E2 -5942.402} C_VEL
LIN {X 0,Y 502.936,Z 724.64,A -85,B 0,C 180,E1 -5945.614,E2 -5945.614} C_VEL
LIN {X 0,Y 502.903,Z 724.639,A -85,B 0,C 180,E1 -5948.033,E2 -5948.033} C_VEL
LIN {X 0,Y 502.88,Z 724.653,A -85,B 0,C 180,E1 -5951.283,E2 -5951.283} C_VEL
LIN {X 0,Y 502.847,Z 724.66,A -85,B 0,C 180,E1 -5954.571,E2 -5954.571} C_VEL
LIN {X 0,Y 502.825,Z 724.651,A -85,B 0,C 180,E1 -5957.908,E2 -5957.908} C_VEL
LIN {X 0,Y 502.831,Z 724.659,A -85,B 0,C 180,E1 -5960.536,E2 -5960.536} C_VEL
LIN {X 0,Y 502.79,Z 724.669,A -85,B 0,C 180,E1 -5963.041,E2 -5963.041} C_VEL
LIN {X 0,Y 502.829,Z 724.651,A -85,B 0,C 180,E1 -5965.676,E2 -5965.676} C_VEL
LIN {X 0,Y 502.841,Z 724.655,A -85,B 0,C 180,E1 -5968.373,E2 -5968.373} C_VEL
LIN {X 0,Y 502.793,Z 724.664,A -85,B 0,C 180,E1 -5971.499,E2 -5971.499} C_VEL
LIN {X 0,Y 502.791,Z 724.659,A -85,B 0,C 180,E1 -5973.995,E2 -5973.995} C_VEL
LIN {X 0,Y 502.779,Z 724.672,A -85,B 0,C 180,E1 -5977.178,E2 -5977.178} C_VEL
LIN {X 0,Y 502.789,Z 724.657,A -85,B 0,C 180,E1 -5980.015,E2 -5980.015} C_VEL
LIN {X 0,Y 502.804,Z 724.641,A -85,B 0,C 180,E1 -5982.199,E2 -5982.199} C_VEL
LIN {X 0,Y 502.787,Z 724.666,A -85,B 0,C 180,E1 -5985.47,E2 -5985.47} C_VEL
LIN {X 0,Y 502.821,Z 724.66,A -85,B 0,C 180,E1 -5988.934,E2 -5988.934} C_VEL
LIN {X 0,Y 502.794,Z 724.66,A -85,B 0,C 180,E1 -5992.046,E2 -5992.046} C_VEL
LIN {X 0,Y 502.797,Z 724.665,A -85,B 0,C 180,E1 -5995.034,E2 -5995.034} C_VEL
LIN {X 0,Y 502.808,Z 724.66,A -85,B 0,C 180,E1 -5997.22,E2 -5997.22} C_VEL
LIN {X 0,Y 502.107,Z 724.749,A -85,B 0,C 180,E1 -5997.888,E2 -5997.888} C_VEL
LIN {X 0,Y 499.246,Z 725.103,A -85,B 0,C 180,E1 -5998.974,E2 -5998.974} C_VEL
LIN {X 0,Y 496.848,Z 725.411,A -85,B 0,C 180,E1 -5999.849,E2 -5999.849} C_VEL
LIN {X 0,Y 495.821,Z 725.533,A -85,B 0,C 180,E1 -6000.525,E2 -6000.525} C_VEL
LIN {X 0,Y 495.737,Z 725.542,A -85,B 0,C 180,E1 -6000.753,E2 -6000.753} C_VEL
LIN {X 0,Y 495.757,Z 725.546,A -85,B 0,C 180,E1 -6003.93,E2 -6003.93} C_VEL
LIN {X 0,Y 495.76,Z 725.539,A -85,B 0,C 180,E1 -6007.14,E2 -6007.14} C_VEL
LIN {X 0,Y 495.785,Z 725.542,A -85,B 0,C 180,E1 -6010.11,E2 -6010.11} C_VEL
LIN {X 0,Y 495.904,Z 725.727,A -85,B 0,C 180,E1 -6011.025,E2 -6011.025} C_VEL
LIN {X 0,Y 496.166,Z 730.675,A -85,B 0,C 180,E1 -6012.27,E2 -6012.27} C_VEL
LIN {X 0,Y 495.76,Z 744.527,A -85,B 0,C 180,E1 -6015.636,E2 -6015.636} C_VEL
LIN {X 0,Y 495.612,Z 752.183,A -85,B 0,C 180,E1 -6017.418,E2 -6017.418} C_VEL
LIN {X 0,Y 496.082,Z 755.264,A -85,B 0,C 180,E1 -6017.522,E2 -6017.522} C_VEL
LIN {X 0,Y 497.242,Z 763.109,A -85,B 0,C 180,E1 -6017.666,E2 -6017.666} C_VEL
LIN {X 0,Y 496.951,Z 827.176,A -85,B 0,C 180,E1 -6018.606,E2 -6018.606} C_VEL
LIN {X 0,Y 496.84,Z 836.321,A -85,B 0,C 180,E1 -6018.836,E2 -6018.836} C_VEL
LIN {X 0,Y 496.643,Z 845.934,A -85,B 0,C 180,E1 -6019.193,E2 -6019.193} C_VEL
LIN {X 0,Y 496.489,Z 855.981,A -85,B 0,C 180,E1 -6019.705,E2 -6019.705} C_VEL
LIN {X 0,Y 496.195,Z 866.408,A -85,B 0,C 180,E1 -6020.42,E2 -6020.42} C_VEL
LIN {X 0,Y 495.901,Z 874.552,A -85,B 0,C 180,E1 -6021.134,E2 -6021.134} C_VEL
LIN {X 0,Y 495.689,Z 881.269,A -85,B 0,C 180,E1 -6021.849,E2 -6021.849} C_VEL
LIN {X 0,Y 495.513,Z 887.625,A -85,B 0,C 180,E1 -6022.666,E2 -6022.666} C_VEL
LIN {X 0,Y 495.418,Z 892.906,A -85,B 0,C 180,E1 -6023.484,E2 -6023.484} C_VEL
LIN {X 0,Y 495.292,Z 897.316,A -85,B 0,C 180,E1 -6024.3,E2 -6024.3} C_VEL
LIN {X 0,Y 495.079,Z 900.993,A -85,B 0,C 180,E1 -6025.114,E2 -6025.114} C_VEL
LIN {X 0,Y 495.188,Z 903.985,A -85,B 0,C 180,E1 -6025.931,E2 -6025.931} C_VEL
LIN {X 0,Y 495.06,Z 906.311,A -85,B 0,C 180,E1 -6026.745,E2 -6026.745} C_VEL
LIN {X 0,Y 495.027,Z 908.081,A -85,B 0,C 180,E1 -6027.559,E2 -6027.559} C_VEL
LIN {X 0,Y 494.962,Z 909.359,A -85,B 0,C 180,E1 -6028.373,E2 -6028.373} C_VEL
LIN {X 0,Y 494.908,Z 910.17,A -85,B 0,C 180,E1 -6029.186,E2 -6029.186} C_VEL
LIN {X 0,Y 494.896,Z 910.478,A -85,B 0,C 180,E1 -6030,E2 -6030} C_VEL
LIN {X 0,Y 494.908,Z 910.206,A -85,B 0,C 180,E1 -6030.814,E2 -6030.814} C_VEL
LIN {X 0,Y 494.963,Z 909.466,A -85,B 0,C 180,E1 -6031.627,E2 -6031.627} C_VEL
LIN {X 0,Y 495.027,Z 908.26,A -85,B 0,C 180,E1 -6032.441,E2 -6032.441} C_VEL
LIN {X 0,Y 495.102,Z 905.418,A -85,B 0,C 180,E1 -6033.662,E2 -6033.662} C_VEL
LIN {X 0,Y 495.162,Z 902.833,A -85,B 0,C 180,E1 -6034.477,E2 -6034.477} C_VEL
LIN {X 0,Y 495.155,Z 899.643,A -85,B 0,C 180,E1 -6035.294,E2 -6035.294} C_VEL
LIN {X 0,Y 495.406,Z 894.591,A -85,B 0,C 180,E1 -6036.312,E2 -6036.312} C_VEL
LIN {X 0,Y 495.446,Z 889.663,A -85,B 0,C 180,E1 -6037.13,E2 -6037.13} C_VEL
LIN {X 0,Y 495.611,Z 883.707,A -85,B 0,C 180,E1 -6037.947,E2 -6037.947} C_VEL
LIN {X 0,Y 495.839,Z 876.456,A -85,B 0,C 180,E1 -6038.764,E2 -6038.764} C_VEL
LIN {X 0,Y 496.102,Z 868.706,A -85,B 0,C 180,E1 -6039.479,E2 -6039.479} C_VEL
LIN {X 0,Y 496.298,Z 860.534,A -85,B 0,C 180,E1 -6040.093,E2 -6040.093} C_VEL
LIN {X 0,Y 496.556,Z 852.005,A -85,B 0,C 180,E1 -6040.603,E2 -6040.603} C_VEL
LIN {X 0,Y 496.814,Z 840.736,A -85,B 0,C 180,E1 -6041.113,E2 -6041.113} C_VEL
LIN {X 0,Y 496.963,Z 829.316,A -85,B 0,C 180,E1 -6041.441,E2 -6041.441} C_VEL
LIN {X 0,Y 497.101,Z 804.795,A -85,B 0,C 180,E1 -6041.824,E2 -6041.824} C_VEL
LIN {X 0,Y 497.095,Z 761.917,A -85,B 0,C 180,E1 -6042.445,E2 -6042.445} C_VEL
LIN {X 0,Y 495.573,Z 752.07,A -85,B 0,C 180,E1 -6042.645,E2 -6042.645} C_VEL
LIN {X 0,Y 495.902,Z 739.699,A -85,B 0,C 180,E1 -6045.621,E2 -6045.621} C_VEL
LIN {X 0,Y 496.153,Z 728.466,A -85,B 0,C 180,E1 -6048.367,E2 -6048.367} C_VEL
LIN {X 0,Y 495.839,Z 725.619,A -85,B 0,C 180,E1 -6049.134,E2 -6049.134} C_VEL
LIN {X 0,Y 495.744,Z 725.543,A -85,B 0,C 180,E1 -6051.629,E2 -6051.629} C_VEL
LIN {X 0,Y 495.716,Z 725.551,A -85,B 0,C 180,E1 -6054.277,E2 -6054.277} C_VEL
LIN {X 0,Y 495.737,Z 725.543,A -85,B 0,C 180,E1 -6056.979,E2 -6056.979} C_VEL
LIN {X 0,Y 495.765,Z 725.545,A -85,B 0,C 180,E1 -6060.147,E2 -6060.147} C_VEL
LIN {X 0,Y 495.79,Z 725.535,A -85,B 0,C 180,E1 -6063.244,E2 -6063.244} C_VEL
LIN {X 0,Y 495.721,Z 725.549,A -85,B 0,C 180,E1 -6066.088,E2 -6066.088} C_VEL
LIN {X 0,Y 495.761,Z 725.536,A -85,B 0,C 180,E1 -6068.768,E2 -6068.768} C_VEL
LIN {X 0,Y 495.757,Z 725.539,A -85,B 0,C 180,E1 -6071.781,E2 -6071.781} C_VEL
LIN {X 0,Y 495.738,Z 725.536,A -85,B 0,C 180,E1 -6075.141,E2 -6075.141} C_VEL
LIN {X 0,Y 495.757,Z 725.521,A -85,B 0,C 180,E1 -6078.219,E2 -6078.219} C_VEL
LIN {X 0,Y 495.751,Z 725.539,A -85,B 0,C 180,E1 -6081.408,E2 -6081.408} C_VEL
LIN {X 0,Y 495.748,Z 725.544,A -85,B 0,C 180,E1 -6084.462,E2 -6084.462} C_VEL
LIN {X 0,Y 495.767,Z 725.536,A -85,B 0,C 180,E1 -6087.406,E2 -6087.406} C_VEL
LIN {X 0,Y 495.767,Z 725.538,A -85,B 0,C 180,E1 -6090.254,E2 -6090.254} C_VEL
LIN {X 0,Y 495.825,Z 725.528,A -85,B 0,C 180,E1 -6093.251,E2 -6093.251} C_VEL
LIN {X 0,Y 495.748,Z 725.538,A -85,B 0,C 180,E1 -6095.725,E2 -6095.725} C_VEL
LIN {X 0,Y 495.744,Z 725.541,A -85,B 0,C 180,E1 -6098.371,E2 -6098.371} C_VEL
LIN {X 0,Y 495.784,Z 725.54,A -85,B 0,C 180,E1 -6100.971,E2 -6100.971} C_VEL
LIN {X 0,Y 495.809,Z 725.527,A -85,B 0,C 180,E1 -6104.376,E2 -6104.376} C_VEL
LIN {X 0,Y 495.787,Z 725.538,A -85,B 0,C 180,E1 -6106.891,E2 -6106.891} C_VEL
LIN {X 0,Y 495.777,Z 725.541,A -85,B 0,C 180,E1 -6109.38,E2 -6109.38} C_VEL
LIN {X 0,Y 495.874,Z 725.515,A -85,B 0,C 180,E1 -6111.852,E2 -6111.852} C_VEL
LIN {X 0,Y 495.892,Z 725.518,A -85,B 0,C 180,E1 -6114.306,E2 -6114.306} C_VEL
LIN {X 0,Y 495.997,Z 725.516,A -85,B 0,C 180,E1 -6117.564,E2 -6117.564} C_VEL
LIN {X 0,Y 496.001,Z 725.506,A -85,B 0,C 180,E1 -6120,E2 -6120} C_VEL
LIN {X 0,Y 495.995,Z 725.498,A -85,B 0,C 180,E1 -6122.436,E2 -6122.436} C_VEL
LIN {X 0,Y 495.893,Z 725.529,A -85,B 0,C 180,E1 -6125.693,E2 -6125.693} C_VEL
LIN {X 0,Y 495.875,Z 725.526,A -85,B 0,C 180,E1 -6128.148,E2 -6128.148} C_VEL
LIN {X 0,Y 495.854,Z 725.526,A -85,B 0,C 180,E1 -6131.445,E2 -6131.445} C_VEL
LIN {X 0,Y 495.792,Z 725.532,A -85,B 0,C 180,E1 -6134.783,E2 -6134.783} C_VEL
LIN {X 0,Y 495.79,Z 725.536,A -85,B 0,C 180,E1 -6137.318,E2 -6137.318} C_VEL
LIN {X 0,Y 495.781,Z 725.538,A -85,B 0,C 180,E1 -6139.89,E2 -6139.89} C_VEL
LIN {X 0,Y 495.767,Z 725.534,A -85,B 0,C 180,E1 -6142.862,E2 -6142.862} C_VEL
LIN {X 0,Y 495.793,Z 725.542,A -85,B 0,C 180,E1 -6146.068,E2 -6146.068} C_VEL
LIN {X 0,Y 495.774,Z 725.531,A -85,B 0,C 180,E1 -6148.815,E2 -6148.815} C_VEL
LIN {X 0,Y 495.758,Z 725.54,A -85,B 0,C 180,E1 -6151.725,E2 -6151.725} C_VEL
LIN {X 0,Y 495.778,Z 725.536,A -85,B 0,C 180,E1 -6154.695,E2 -6154.695} C_VEL
LIN {X 0,Y 495.733,Z 725.532,A -85,B 0,C 180,E1 -6157.561,E2 -6157.561} C_VEL
LIN {X 0,Y 495.781,Z 725.531,A -85,B 0,C 180,E1 -6160.698,E2 -6160.698} C_VEL
LIN {X 0,Y 495.735,Z 725.544,A -85,B 0,C 180,E1 -6164.001,E2 -6164.001} C_VEL
LIN {X 0,Y 495.727,Z 725.539,A -85,B 0,C 180,E1 -6167.117,E2 -6167.117} C_VEL
LIN {X 0,Y 495.761,Z 725.536,A -85,B 0,C 180,E1 -6169.953,E2 -6169.953} C_VEL
LIN {X 0,Y 495.732,Z 725.549,A -85,B 0,C 180,E1 -6172.552,E2 -6172.552} C_VEL
LIN {X 0,Y 495.786,Z 725.536,A -85,B 0,C 180,E1 -6175.457,E2 -6175.457} C_VEL
LIN {X 0,Y 495.76,Z 725.54,A -85,B 0,C 180,E1 -6178.364,E2 -6178.364} C_VEL
LIN {X 0,Y 495.789,Z 725.537,A -85,B 0,C 180,E1 -6181.507,E2 -6181.507} C_VEL
LIN {X 0,Y 495.791,Z 725.535,A -85,B 0,C 180,E1 -6183.932,E2 -6183.932} C_VEL
LIN {X 0,Y 495.794,Z 725.583,A -85,B 0,C 180,E1 -6186.831,E2 -6186.831} C_VEL
LIN {X 0,Y 496.95,Z 733.033,A -85,B 0,C 180,E1 -6188.426,E2 -6188.426} C_VEL
LIN {X 0,Y 496.468,Z 748.807,A -85,B 0,C 180,E1 -6191.523,E2 -6191.523} C_VEL
LIN {X 0,Y 496.03,Z 764.014,A -85,B 0,C 180,E1 -6194.463,E2 -6194.463} C_VEL
LIN {X 0,Y 495.717,Z 779.188,A -85,B 0,C 180,E1 -6197.353,E2 -6197.353} C_VEL
LIN {X 0,Y 495.915,Z 781.343,A -85,B 0,C 180,E1 -6197.437,E2 -6197.437} C_VEL
LIN {X 0,Y 497.19,Z 792.331,A -85,B 0,C 180,E1 -6197.629,E2 -6197.629} C_VEL
LIN {X 0,Y 496.945,Z 856.8,A -85,B 0,C 180,E1 -6198.58,E2 -6198.58} C_VEL
LIN {X 0,Y 496.737,Z 866.444,A -85,B 0,C 180,E1 -6198.834,E2 -6198.834} C_VEL
LIN {X 0,Y 496.52,Z 877.996,A -85,B 0,C 180,E1 -6199.293,E2 -6199.293} C_VEL
LIN {X 0,Y 496.28,Z 888.633,A -85,B 0,C 180,E1 -6199.907,E2 -6199.907} C_VEL
LIN {X 0,Y 496.03,Z 896.962,A -85,B 0,C 180,E1 -6200.52,E2 -6200.52} C_VEL
LIN {X 0,Y 495.753,Z 904.844,A -85,B 0,C 180,E1 -6201.234,E2 -6201.234} C_VEL
LIN {X 0,Y 495.569,Z 912.217,A -85,B 0,C 180,E1 -6202.052,E2 -6202.052} C_VEL
LIN {X 0,Y 495.378,Z 919.966,A -85,B 0,C 180,E1 -6203.115,E2 -6203.115} C_VEL
LIN {X 0,Y 495.239,Z 926.529,A -85,B 0,C 180,E1 -6204.299,E2 -6204.299} C_VEL
LIN {X 0,Y 495.08,Z 931.713,A -85,B 0,C 180,E1 -6205.522,E2 -6205.522} C_VEL
LIN {X 0,Y 495.096,Z 934.366,A -85,B 0,C 180,E1 -6206.338,E2 -6206.338} C_VEL
LIN {X 0,Y 494.976,Z 937.272,A -85,B 0,C 180,E1 -6207.559,E2 -6207.559} C_VEL
LIN {X 0,Y 494.959,Z 938.528,A -85,B 0,C 180,E1 -6208.373,E2 -6208.373} C_VEL
LIN {X 0,Y 494.908,Z 939.308,A -85,B 0,C 180,E1 -6209.186,E2 -6209.186} C_VEL
LIN {X 0,Y 494.895,Z 939.604,A -85,B 0,C 180,E1 -6210,E2 -6210} C_VEL
LIN {X 0,Y 494.908,Z 939.308,A -85,B 0,C 180,E1 -6210.814,E2 -6210.814} C_VEL
LIN {X 0,Y 494.959,Z 938.527,A -85,B 0,C 180,E1 -6211.627,E2 -6211.627} C_VEL
LIN {X 0,Y 494.976,Z 937.271,A -85,B 0,C 180,E1 -6212.441,E2 -6212.441} C_VEL
LIN {X 0,Y 495.096,Z 934.365,A -85,B 0,C 180,E1 -6213.662,E2 -6213.662} C_VEL
LIN {X 0,Y 495.08,Z 931.713,A -85,B 0,C 180,E1 -6214.478,E2 -6214.478} C_VEL
LIN {X 0,Y 495.239,Z 926.526,A -85,B 0,C 180,E1 -6215.701,E2 -6215.701} C_VEL
LIN {X 0,Y 495.38,Z 919.96,A -85,B 0,C 180,E1 -6216.885,E2 -6216.885} C_VEL
LIN {X 0,Y 495.568,Z 912.219,A -85,B 0,C 180,E1 -6217.948,E2 -6217.948} C_VEL
LIN {X 0,Y 495.753,Z 904.851,A -85,B 0,C 180,E1 -6218.766,E2 -6218.766} C_VEL
LIN {X 0,Y 496.03,Z 896.965,A -85,B 0,C 180,E1 -6219.48,E2 -6219.48} C_VEL
LIN {X 0,Y 496.28,Z 888.634,A -85,B 0,C 180,E1 -6220.093,E2 -6220.093} C_VEL
LIN {X 0,Y 496.531,Z 878,A -85,B 0,C 180,E1 -6220.706,E2 -6220.706} C_VEL
LIN {X 0,Y 496.771,Z 866.449,A -85,B 0,C 180,E1 -6221.165,E2 -6221.165} C_VEL
LIN {X 0,Y 496.944,Z 856.802,A -85,B 0,C 180,E1 -6221.42,E2 -6221.42} C_VEL
LIN {X 0,Y 497.149,Z 805.441,A -85,B 0,C 180,E1 -6222.183,E2 -6222.183} C_VEL
LIN {X 0,Y 497.018,Z 789.47,A -85,B 0,C 180,E1 -6222.417,E2 -6222.417} C_VEL
LIN {X 0,Y 495.728,Z 779.444,A -85,B 0,C 180,E1 -6222.621,E2 -6222.621} C_VEL
LIN {X 0,Y 495.997,Z 765.919,A -85,B 0,C 180,E1 -6225.162,E2 -6225.162} C_VEL
LIN {X 0,Y 496.351,Z 751.587,A -85,B 0,C 180,E1 -6227.937,E2 -6227.937} C_VEL
LIN {X 0,Y 496.834,Z 737.404,A -85,B 0,C 180,E1 -6230.71,E2 -6230.71} C_VEL
LIN {X 0,Y 496.888,Z 731.943,A -85,B 0,C 180,E1 -6231.795,E2 -6231.795} C_VEL
LIN {X 0,Y 495.794,Z 725.584,A -85,B 0,C 180,E1 -6233.169,E2 -6233.169} C_VEL
LIN {X 0,Y 495.791,Z 725.534,A -85,B 0,C 180,E1 -6236.068,E2 -6236.068} C_VEL
LIN {X 0,Y 495.773,Z 725.542,A -85,B 0,C 180,E1 -6238.815,E2 -6238.815} C_VEL
LIN {X 0,Y 495.76,Z 725.541,A -85,B 0,C 180,E1 -6241.726,E2 -6241.726} C_VEL
LIN {X 0,Y 495.778,Z 725.538,A -85,B 0,C 180,E1 -6244.695,E2 -6244.695} C_VEL
LIN {X 0,Y 495.733,Z 725.55,A -85,B 0,C 180,E1 -6247.561,E2 -6247.561} C_VEL
LIN {X 0,Y 495.768,Z 725.533,A -85,B 0,C 180,E1 -6250.7,E2 -6250.7} C_VEL
LIN {X 0,Y 495.735,Z 725.545,A -85,B 0,C 180,E1 -6254.001,E2 -6254.001} C_VEL
LIN {X 0,Y 495.727,Z 725.543,A -85,B 0,C 180,E1 -6257.117,E2 -6257.117} C_VEL
LIN {X 0,Y 495.79,Z 725.517,A -85,B 0,C 180,E1 -6259.949,E2 -6259.949} C_VEL
LIN {X 0,Y 495.732,Z 725.533,A -85,B 0,C 180,E1 -6262.553,E2 -6262.553} C_VEL
LIN {X 0,Y 495.787,Z 725.537,A -85,B 0,C 180,E1 -6265.458,E2 -6265.458} C_VEL
LIN {X 0,Y 495.758,Z 725.539,A -85,B 0,C 180,E1 -6268.364,E2 -6268.364} C_VEL
LIN {X 0,Y 495.789,Z 725.532,A -85,B 0,C 180,E1 -6271.507,E2 -6271.507} C_VEL
LIN {X 0,Y 495.793,Z 725.542,A -85,B 0,C 180,E1 -6273.932,E2 -6273.932} C_VEL
LIN {X 0,Y 495.767,Z 725.534,A -85,B 0,C 180,E1 -6277.138,E2 -6277.138} C_VEL
LIN {X 0,Y 495.781,Z 725.538,A -85,B 0,C 180,E1 -6280.11,E2 -6280.11} C_VEL
LIN {X 0,Y 495.79,Z 725.537,A -85,B 0,C 180,E1 -6282.682,E2 -6282.682} C_VEL
LIN {X 0,Y 495.792,Z 725.532,A -85,B 0,C 180,E1 -6285.217,E2 -6285.217} C_VEL
LIN {X 0,Y 495.854,Z 725.527,A -85,B 0,C 180,E1 -6288.555,E2 -6288.555} C_VEL
LIN {X 0,Y 495.876,Z 725.526,A -85,B 0,C 180,E1 -6291.852,E2 -6291.852} C_VEL
LIN {X 0,Y 495.894,Z 725.529,A -85,B 0,C 180,E1 -6294.307,E2 -6294.307} C_VEL
LIN {X 0,Y 495.996,Z 725.498,A -85,B 0,C 180,E1 -6297.564,E2 -6297.564} C_VEL
LIN {X 0,Y 496.001,Z 725.506,A -85,B 0,C 180,E1 -6300,E2 -6300} C_VEL
LIN {X 0,Y 495.997,Z 725.515,A -85,B 0,C 180,E1 -6302.436,E2 -6302.436} C_VEL
LIN {X 0,Y 495.892,Z 725.517,A -85,B 0,C 180,E1 -6305.694,E2 -6305.694} C_VEL
LIN {X 0,Y 495.874,Z 725.515,A -85,B 0,C 180,E1 -6308.148,E2 -6308.148} C_VEL
LIN {X 0,Y 495.854,Z 725.527,A -85,B 0,C 180,E1 -6311.445,E2 -6311.445} C_VEL
LIN {X 0,Y 495.792,Z 725.54,A -85,B 0,C 180,E1 -6314.783,E2 -6314.783} C_VEL
LIN {X 0,Y 495.767,Z 725.533,A -85,B 0,C 180,E1 -6317.319,E2 -6317.319} C_VEL
LIN {X 0,Y 495.773,Z 725.535,A -85,B 0,C 180,E1 -6319.89,E2 -6319.89} C_VEL
LIN {X 0,Y 495.761,Z 725.546,A -85,B 0,C 180,E1 -6322.86,E2 -6322.86} C_VEL
LIN {X 0,Y 495.785,Z 725.527,A -85,B 0,C 180,E1 -6326.068,E2 -6326.068} C_VEL
LIN {X 0,Y 495.773,Z 725.54,A -85,B 0,C 180,E1 -6328.815,E2 -6328.815} C_VEL
LIN {X 0,Y 495.756,Z 725.538,A -85,B 0,C 180,E1 -6331.725,E2 -6331.725} C_VEL
LIN {X 0,Y 495.764,Z 725.536,A -85,B 0,C 180,E1 -6334.693,E2 -6334.693} C_VEL
LIN {X 0,Y 495.73,Z 725.546,A -85,B 0,C 180,E1 -6337.562,E2 -6337.562} C_VEL
LIN {X 0,Y 495.768,Z 725.531,A -85,B 0,C 180,E1 -6340.7,E2 -6340.7} C_VEL
LIN {X 0,Y 495.726,Z 725.537,A -85,B 0,C 180,E1 -6344.002,E2 -6344.002} C_VEL
LIN {X 0,Y 495.726,Z 725.546,A -85,B 0,C 180,E1 -6347.117,E2 -6347.117} C_VEL
LIN {X 0,Y 495.76,Z 725.536,A -85,B 0,C 180,E1 -6349.953,E2 -6349.953} C_VEL
LIN {X 0,Y 495.729,Z 725.537,A -85,B 0,C 180,E1 -6352.553,E2 -6352.553} C_VEL
LIN {X 0,Y 495.772,Z 725.545,A -85,B 0,C 180,E1 -6355.456,E2 -6355.456} C_VEL
LIN {X 0,Y 495.756,Z 725.536,A -85,B 0,C 180,E1 -6358.364,E2 -6358.364} C_VEL
LIN {X 0,Y 495.737,Z 725.542,A -85,B 0,C 180,E1 -6360.753,E2 -6360.753} C_VEL
LIN {X 0,Y 495.066,Z 725.631,A -85,B 0,C 180,E1 -6361.432,E2 -6361.432} C_VEL
LIN {X 0,Y 492.2,Z 725.984,A -85,B 0,C 180,E1 -6362.534,E2 -6362.534} C_VEL
LIN {X 0,Y 489.791,Z 726.287,A -85,B 0,C 180,E1 -6363.422,E2 -6363.422} C_VEL
LIN {X 0,Y 488.776,Z 726.414,A -85,B 0,C 180,E1 -6364.109,E2 -6364.109} C_VEL
LIN {X 0,Y 488.704,Z 726.42,A -85,B 0,C 180,E1 -6364.341,E2 -6364.341} C_VEL
LIN {X 0,Y 488.723,Z 726.415,A -85,B 0,C 180,E1 -6367.153,E2 -6367.153} C_VEL
LIN {X 0,Y 488.734,Z 726.422,A -85,B 0,C 180,E1 -6369.811,E2 -6369.811} C_VEL
LIN {X 0,Y 488.81,Z 726.576,A -85,B 0,C 180,E1 -6370.908,E2 -6370.908} C_VEL
LIN {X 0,Y 489.147,Z 730.836,A -85,B 0,C 180,E1 -6372.006,E2 -6372.006} C_VEL
LIN {X 0,Y 488.807,Z 742.957,A -85,B 0,C 180,E1 -6375.001,E2 -6375.001} C_VEL
LIN {X 0,Y 488.582,Z 752.388,A -85,B 0,C 180,E1 -6377.236,E2 -6377.236} C_VEL
LIN {X 0,Y 489.15,Z 756.065,A -85,B 0,C 180,E1 -6377.35,E2 -6377.35} C_VEL
LIN {X 0,Y 490.299,Z 763.948,A -85,B 0,C 180,E1 -6377.497,E2 -6377.497} C_VEL
LIN {X 0,Y 490.02,Z 827.416,A -85,B 0,C 180,E1 -6378.443,E2 -6378.443} C_VEL
LIN {X 0,Y 489.9,Z 836.549,A -85,B 0,C 180,E1 -6378.676,E2 -6378.676} C_VEL
LIN {X 0,Y 489.689,Z 846.156,A -85,B 0,C 180,E1 -6379.038,E2 -6379.038} C_VEL
LIN {X 0,Y 489.503,Z 856.201,A -85,B 0,C 180,E1 -6379.557,E2 -6379.557} C_VEL
LIN {X 0,Y 489.192,Z 866.624,A -85,B 0,C 180,E1 -6380.282,E2 -6380.282} C_VEL
LIN {X 0,Y 488.91,Z 874.766,A -85,B 0,C 180,E1 -6381.006,E2 -6381.006} C_VEL
LIN {X 0,Y 488.657,Z 881.482,A -85,B 0,C 180,E1 -6381.731,E2 -6381.731} C_VEL
LIN {X 0,Y 488.459,Z 887.837,A -85,B 0,C 180,E1 -6382.56,E2 -6382.56} C_VEL
LIN {X 0,Y 488.357,Z 893.117,A -85,B 0,C 180,E1 -6383.389,E2 -6383.389} C_VEL
LIN {X 0,Y 488.249,Z 897.527,A -85,B 0,C 180,E1 -6384.217,E2 -6384.217} C_VEL
LIN {X 0,Y 488.009,Z 901.204,A -85,B 0,C 180,E1 -6385.043,E2 -6385.043} C_VEL
LIN {X 0,Y 488.105,Z 904.195,A -85,B 0,C 180,E1 -6385.872,E2 -6385.872} C_VEL
LIN {X 0,Y 487.989,Z 906.519,A -85,B 0,C 180,E1 -6386.697,E2 -6386.697} C_VEL
LIN {X 0,Y 487.936,Z 908.29,A -85,B 0,C 180,E1 -6387.523,E2 -6387.523} C_VEL
LIN {X 0,Y 487.891,Z 909.568,A -85,B 0,C 180,E1 -6388.349,E2 -6388.349} C_VEL
LIN {X 0,Y 487.831,Z 910.378,A -85,B 0,C 180,E1 -6389.175,E2 -6389.175} C_VEL
LIN {X 0,Y 487.817,Z 910.686,A -85,B 0,C 180,E1 -6390,E2 -6390} C_VEL
LIN {X 0,Y 487.832,Z 910.413,A -85,B 0,C 180,E1 -6390.825,E2 -6390.825} C_VEL
LIN {X 0,Y 487.892,Z 909.673,A -85,B 0,C 180,E1 -6391.651,E2 -6391.651} C_VEL
LIN {X 0,Y 487.936,Z 908.466,A -85,B 0,C 180,E1 -6392.477,E2 -6392.477} C_VEL
LIN {X 0,Y 488.036,Z 905.624,A -85,B 0,C 180,E1 -6393.716,E2 -6393.716} C_VEL
LIN {X 0,Y 488.073,Z 903.039,A -85,B 0,C 180,E1 -6394.542,E2 -6394.542} C_VEL
LIN {X 0,Y 488.101,Z 899.848,A -85,B 0,C 180,E1 -6395.37,E2 -6395.37} C_VEL
LIN {X 0,Y 488.338,Z 894.366,A -85,B 0,C 180,E1 -6396.48,E2 -6396.48} C_VEL
LIN {X 0,Y 488.396,Z 890.006,A -85,B 0,C 180,E1 -6397.213,E2 -6397.213} C_VEL
LIN {X 0,Y 488.584,Z 883.909,A -85,B 0,C 180,E1 -6398.062,E2 -6398.062} C_VEL
LIN {X 0,Y 488.841,Z 876.657,A -85,B 0,C 180,E1 -6398.891,E2 -6398.891} C_VEL
LIN {X 0,Y 489.095,Z 868.906,A -85,B 0,C 180,E1 -6399.616,E2 -6399.616} C_VEL
LIN {X 0,Y 489.319,Z 860.732,A -85,B 0,C 180,E1 -6400.238,E2 -6400.238} C_VEL
LIN {X 0,Y 489.578,Z 852.201,A -85,B 0,C 180,E1 -6400.755,E2 -6400.755} C_VEL
LIN {X 0,Y 489.877,Z 840.926,A -85,B 0,C 180,E1 -6401.272,E2 -6401.272} C_VEL
LIN {X 0,Y 490.017,Z 829.54,A -85,B 0,C 180,E1 -6401.604,E2 -6401.604} C_VEL
LIN {X 0,Y 490.153,Z 806.256,A -85,B 0,C 180,E1 -6401.975,E2 -6401.975} C_VEL
LIN {X 0,Y 490.213,Z 762.896,A -85,B 0,C 180,E1 -6402.611,E2 -6402.611} C_VEL
LIN {X 0,Y 488.527,Z 752.285,A -85,B 0,C 180,E1 -6402.825,E2 -6402.825} C_VEL
LIN {X 0,Y 488.886,Z 739.858,A -85,B 0,C 180,E1 -6405.851,E2 -6405.851} C_VEL
LIN {X 0,Y 489.133,Z 729.17,A -85,B 0,C 180,E1 -6408.503,E2 -6408.503} C_VEL
LIN {X 0,Y 488.797,Z 726.485,A -85,B 0,C 180,E1 -6409.257,E2 -6409.257} C_VEL
LIN {X 0,Y 488.699,Z 726.424,A -85,B 0,C 180,E1 -6411.957,E2 -6411.957} C_VEL
LIN {X 0,Y 488.7,Z 726.42,A -85,B 0,C 180,E1 -6415.041,E2 -6415.041} C_VEL
LIN {X 0,Y 488.712,Z 726.423,A -85,B 0,C 180,E1 -6418.331,E2 -6418.331} C_VEL
LIN {X 0,Y 488.692,Z 726.415,A -85,B 0,C 180,E1 -6421.18,E2 -6421.18} C_VEL
LIN {X 0,Y 488.725,Z 726.419,A -85,B 0,C 180,E1 -6424.113,E2 -6424.113} C_VEL
LIN {X 0,Y 488.68,Z 726.416,A -85,B 0,C 180,E1 -6427.159,E2 -6427.159} C_VEL
LIN {X 0,Y 488.72,Z 726.415,A -85,B 0,C 180,E1 -6430.345,E2 -6430.345} C_VEL
LIN {X 0,Y 488.685,Z 726.419,A -85,B 0,C 180,E1 -6433.655,E2 -6433.655} C_VEL
LIN {X 0,Y 488.68,Z 726.415,A -85,B 0,C 180,E1 -6436.345,E2 -6436.345} C_VEL
LIN {X 0,Y 488.735,Z 726.405,A -85,B 0,C 180,E1 -6439.677,E2 -6439.677} C_VEL
LIN {X 0,Y 488.68,Z 726.429,A -85,B 0,C 180,E1 -6442.841,E2 -6442.841} C_VEL
LIN {X 0,Y 488.725,Z 726.411,A -85,B 0,C 180,E1 -6445.887,E2 -6445.887} C_VEL
LIN {X 0,Y 488.693,Z 726.423,A -85,B 0,C 180,E1 -6448.82,E2 -6448.82} C_VEL
LIN {X 0,Y 488.744,Z 726.412,A -85,B 0,C 180,E1 -6451.671,E2 -6451.671} C_VEL
LIN {X 0,Y 488.741,Z 726.406,A -85,B 0,C 180,E1 -6454.444,E2 -6454.444} C_VEL
LIN {X 0,Y 488.724,Z 726.423,A -85,B 0,C 180,E1 -6457.153,E2 -6457.153} C_VEL
LIN {X 0,Y 488.727,Z 726.414,A -85,B 0,C 180,E1 -6459.81,E2 -6459.81} C_VEL
LIN {X 0,Y 488.717,Z 726.408,A -85,B 0,C 180,E1 -6462.423,E2 -6462.423} C_VEL
LIN {X 0,Y 488.767,Z 726.41,A -85,B 0,C 180,E1 -6465,E2 -6465} C_VEL
LIN {X 0,Y 488.808,Z 726.404,A -85,B 0,C 180,E1 -6468.388,E2 -6468.388} C_VEL
LIN {X 0,Y 488.818,Z 726.395,A -85,B 0,C 180,E1 -6471.734,E2 -6471.734} C_VEL
LIN {X 0,Y 488.85,Z 726.395,A -85,B 0,C 180,E1 -6474.224,E2 -6474.224} C_VEL
LIN {X 0,Y 488.964,Z 726.393,A -85,B 0,C 180,E1 -6477.529,E2 -6477.529} C_VEL
LIN {X 0,Y 488.972,Z 726.381,A -85,B 0,C 180,E1 -6480,E2 -6480} C_VEL
LIN {X 0,Y 488.963,Z 726.374,A -85,B 0,C 180,E1 -6482.471,E2 -6482.471} C_VEL
LIN {X 0,Y 488.851,Z 726.406,A -85,B 0,C 180,E1 -6485.776,E2 -6485.776} C_VEL
LIN {X 0,Y 488.82,Z 726.404,A -85,B 0,C 180,E1 -6488.266,E2 -6488.266} C_VEL
LIN {X 0,Y 488.808,Z 726.403,A -85,B 0,C 180,E1 -6491.612,E2 -6491.612} C_VEL
LIN {X 0,Y 488.764,Z 726.408,A -85,B 0,C 180,E1 -6495,E2 -6495} C_VEL
LIN {X 0,Y 488.757,Z 726.411,A -85,B 0,C 180,E1 -6498.442,E2 -6498.442} C_VEL
LIN {X 0,Y 488.709,Z 726.408,A -85,B 0,C 180,E1 -6501.071,E2 -6501.071} C_VEL
LIN {X 0,Y 488.696,Z 726.42,A -85,B 0,C 180,E1 -6503.745,E2 -6503.745} C_VEL
LIN {X 0,Y 488.794,Z 726.405,A -85,B 0,C 180,E1 -6506.944,E2 -6506.944} C_VEL
LIN {X 0,Y 488.711,Z 726.42,A -85,B 0,C 180,E1 -6510.363,E2 -6510.363} C_VEL
LIN {X 0,Y 488.737,Z 726.414,A -85,B 0,C 180,E1 -6513.484,E2 -6513.484} C_VEL
LIN {X 0,Y 488.691,Z 726.416,A -85,B 0,C 180,E1 -6516.356,E2 -6516.356} C_VEL
LIN {X 0,Y 488.743,Z 726.389,A -85,B 0,C 180,E1 -6519.25,E2 -6519.25} C_VEL
LIN {X 0,Y 488.713,Z 726.408,A -85,B 0,C 180,E1 -6521.6,E2 -6521.6} C_VEL
LIN {X 0,Y 488.713,Z 726.42,A -85,B 0,C 180,E1 -6524.801,E2 -6524.801} C_VEL
LIN {X 0,Y 488.692,Z 726.414,A -85,B 0,C 180,E1 -6527.474,E2 -6527.474} C_VEL
LIN {X 0,Y 488.732,Z 726.42,A -85,B 0,C 180,E1 -6530.749,E2 -6530.749} C_VEL
LIN {X 0,Y 488.686,Z 726.417,A -85,B 0,C 180,E1 -6533.869,E2 -6533.869} C_VEL
LIN {X 0,Y 488.74,Z 726.417,A -85,B 0,C 180,E1 -6536.877,E2 -6536.877} C_VEL
LIN {X 0,Y 488.725,Z 726.408,A -85,B 0,C 180,E1 -6539.781,E2 -6539.781} C_VEL
LIN {X 0,Y 488.793,Z 726.406,A -85,B 0,C 180,E1 -6543.056,E2 -6543.056} C_VEL
LIN {X 0,Y 488.704,Z 726.418,A -85,B 0,C 180,E1 -6546.255,E2 -6546.255} C_VEL
LIN {X 0,Y 488.757,Z 726.574,A -85,B 0,C 180,E1 -6546.745,E2 -6546.745} C_VEL
LIN {X 0,Y 489.955,Z 733.911,A -85,B 0,C 180,E1 -6548.314,E2 -6548.314} C_VEL
LIN {X 0,Y 489.478,Z 749.273,A -85,B 0,C 180,E1 -6551.376,E2 -6551.376} C_VEL
LIN {X 0,Y 488.98,Z 766.118,A -85,B 0,C 180,E1 -6554.682,E2 -6554.682} C_VEL
LIN {X 0,Y 488.642,Z 779.026,A -85,B 0,C 180,E1 -6557.171,E2 -6557.171} C_VEL
LIN {X 0,Y 488.898,Z 781.146,A -85,B 0,C 180,E1 -6557.254,E2 -6557.254} C_VEL
LIN {X 0,Y 490.283,Z 793.505,A -85,B 0,C 180,E1 -6557.472,E2 -6557.472} C_VEL
LIN {X 0,Y 490.005,Z 856.592,A -85,B 0,C 180,E1 -6558.416,E2 -6558.416} C_VEL
LIN {X 0,Y 489.773,Z 867.068,A -85,B 0,C 180,E1 -6558.699,E2 -6558.699} C_VEL
LIN {X 0,Y 489.561,Z 877.788,A -85,B 0,C 180,E1 -6559.139,E2 -6559.139} C_VEL
LIN {X 0,Y 489.271,Z 888.423,A -85,B 0,C 180,E1 -6559.761,E2 -6559.761} C_VEL
LIN {X 0,Y 489.024,Z 896.753,A -85,B 0,C 180,E1 -6560.383,E2 -6560.383} C_VEL
LIN {X 0,Y 488.742,Z 904.636,A -85,B 0,C 180,E1 -6561.107,E2 -6561.107} C_VEL
LIN {X 0,Y 488.519,Z 912.008,A -85,B 0,C 180,E1 -6561.937,E2 -6561.937} C_VEL
LIN {X 0,Y 488.315,Z 919.757,A -85,B 0,C 180,E1 -6563.015,E2 -6563.015} C_VEL
LIN {X 0,Y 488.175,Z 926.32,A -85,B 0,C 180,E1 -6564.216,E2 -6564.216} C_VEL
LIN {X 0,Y 487.984,Z 931.504,A -85,B 0,C 180,E1 -6565.457,E2 -6565.457} C_VEL
LIN {X 0,Y 487.987,Z 935.314,A -85,B 0,C 180,E1 -6566.697,E2 -6566.697} C_VEL
LIN {X 0,Y 487.889,Z 937.064,A -85,B 0,C 180,E1 -6567.523,E2 -6567.523} C_VEL
LIN {X 0,Y 487.887,Z 938.32,A -85,B 0,C 180,E1 -6568.349,E2 -6568.349} C_VEL
LIN {X 0,Y 487.831,Z 939.1,A -85,B 0,C 180,E1 -6569.175,E2 -6569.175} C_VEL
LIN {X 0,Y 487.816,Z 939.395,A -85,B 0,C 180,E1 -6570,E2 -6570} C_VEL
LIN {X 0,Y 487.831,Z 939.1,A -85,B 0,C 180,E1 -6570.825,E2 -6570.825} C_VEL
LIN {X 0,Y 487.887,Z 938.319,A -85,B 0,C 180,E1 -6571.651,E2 -6571.651} C_VEL
LIN {X 0,Y 487.889,Z 937.063,A -85,B 0,C 180,E1 -6572.477,E2 -6572.477} C_VEL
LIN {X 0,Y 488.021,Z 934.157,A -85,B 0,C 180,E1 -6573.716,E2 -6573.716} C_VEL
LIN {X 0,Y 487.984,Z 931.503,A -85,B 0,C 180,E1 -6574.543,E2 -6574.543} C_VEL
LIN {X 0,Y 488.175,Z 926.317,A -85,B 0,C 180,E1 -6575.784,E2 -6575.784} C_VEL
LIN {X 0,Y 488.31,Z 919.751,A -85,B 0,C 180,E1 -6576.985,E2 -6576.985} C_VEL
LIN {X 0,Y 488.519,Z 912.01,A -85,B 0,C 180,E1 -6578.063,E2 -6578.063} C_VEL
LIN {X 0,Y 488.742,Z 904.642,A -85,B 0,C 180,E1 -6578.893,E2 -6578.893} C_VEL
LIN {X 0,Y 489.024,Z 896.756,A -85,B 0,C 180,E1 -6579.617,E2 -6579.617} C_VEL
LIN {X 0,Y 489.271,Z 888.424,A -85,B 0,C 180,E1 -6580.239,E2 -6580.239} C_VEL
LIN {X 0,Y 489.575,Z 877.792,A -85,B 0,C 180,E1 -6580.86,E2 -6580.86} C_VEL
LIN {X 0,Y 489.797,Z 866.239,A -85,B 0,C 180,E1 -6581.326,E2 -6581.326} C_VEL
LIN {X 0,Y 489.995,Z 856.593,A -85,B 0,C 180,E1 -6581.584,E2 -6581.584} C_VEL
LIN {X 0,Y 490.227,Z 809.348,A -85,B 0,C 180,E1 -6582.297,E2 -6582.297} C_VEL
LIN {X 0,Y 490.107,Z 790.285,A -85,B 0,C 180,E1 -6582.58,E2 -6582.58} C_VEL
LIN {X 0,Y 488.661,Z 779.291,A -85,B 0,C 180,E1 -6582.804,E2 -6582.804} C_VEL
LIN {X 0,Y 488.866,Z 770.987,A -85,B 0,C 180,E1 -6584.359,E2 -6584.359} C_VEL
LIN {X 0,Y 489.305,Z 754.685,A -85,B 0,C 180,E1 -6587.555,E2 -6587.555} C_VEL
LIN {X 0,Y 489.824,Z 739.422,A -85,B 0,C 180,E1 -6590.581,E2 -6590.581} C_VEL
LIN {X 0,Y 489.878,Z 732.864,A -85,B 0,C 180,E1 -6591.901,E2 -6591.901} C_VEL
LIN {X 0,Y 488.733,Z 726.469,A -85,B 0,C 180,E1 -6593.305,E2 -6593.305} C_VEL
LIN {X 0,Y 488.757,Z 726.409,A -85,B 0,C 180,E1 -6596.472,E2 -6596.472} C_VEL
LIN {X 0,Y 488.724,Z 726.417,A -85,B 0,C 180,E1 -6599.27,E2 -6599.27} C_VEL
LIN {X 0,Y 488.706,Z 726.416,A -85,B 0,C 180,E1 -6602.147,E2 -6602.147} C_VEL
LIN {X 0,Y 488.724,Z 726.421,A -85,B 0,C 180,E1 -6605.115,E2 -6605.115} C_VEL
LIN {X 0,Y 488.683,Z 726.421,A -85,B 0,C 180,E1 -6608.2,E2 -6608.2} C_VEL
LIN {X 0,Y 488.719,Z 726.411,A -85,B 0,C 180,E1 -6610.345,E2 -6610.345} C_VEL
LIN {X 0,Y 488.688,Z 726.426,A -85,B 0,C 180,E1 -6613.654,E2 -6613.654} C_VEL
LIN {X 0,Y 488.688,Z 726.418,A -85,B 0,C 180,E1 -6616.346,E2 -6616.346} C_VEL
LIN {X 0,Y 488.734,Z 726.399,A -85,B 0,C 180,E1 -6619.677,E2 -6619.677} C_VEL
LIN {X 0,Y 488.682,Z 726.412,A -85,B 0,C 180,E1 -6622.278,E2 -6622.278} C_VEL
LIN {X 0,Y 488.73,Z 726.412,A -85,B 0,C 180,E1 -6625.052,E2 -6625.052} C_VEL
LIN {X 0,Y 488.705,Z 726.421,A -85,B 0,C 180,E1 -6628.046,E2 -6628.046} C_VEL
LIN {X 0,Y 488.725,Z 726.409,A -85,B 0,C 180,E1 -6630.73,E2 -6630.73} C_VEL
LIN {X 0,Y 488.759,Z 726.412,A -85,B 0,C 180,E1 -6633.528,E2 -6633.528} C_VEL
LIN {X 0,Y 488.696,Z 726.42,A -85,B 0,C 180,E1 -6636.255,E2 -6636.255} C_VEL
LIN {X 0,Y 488.748,Z 726.404,A -85,B 0,C 180,E1 -6639.176,E2 -6639.176} C_VEL
LIN {X 0,Y 488.761,Z 726.411,A -85,B 0,C 180,E1 -6641.628,E2 -6641.628} C_VEL
LIN {X 0,Y 488.764,Z 726.408,A -85,B 0,C 180,E1 -6645,E2 -6645} C_VEL
LIN {X 0,Y 488.808,Z 726.403,A -85,B 0,C 180,E1 -6648.388,E2 -6648.388} C_VEL
LIN {X 0,Y 488.82,Z 726.404,A -85,B 0,C 180,E1 -6651.734,E2 -6651.734} C_VEL
LIN {X 0,Y 488.852,Z 726.405,A -85,B 0,C 180,E1 -6654.224,E2 -6654.224} C_VEL
LIN {X 0,Y 488.964,Z 726.373,A -85,B 0,C 180,E1 -6657.529,E2 -6657.529} C_VEL
LIN {X 0,Y 488.957,Z 726.39,A -85,B 0,C 180,E1 -6660.824,E2 -6660.824} C_VEL
LIN {X 0,Y 488.965,Z 726.392,A -85,B 0,C 180,E1 -6662.471,E2 -6662.471} C_VEL
LIN {X 0,Y 488.85,Z 726.395,A -85,B 0,C 180,E1 -6665.776,E2 -6665.776} C_VEL
LIN {X 0,Y 488.818,Z 726.394,A -85,B 0,C 180,E1 -6668.266,E2 -6668.266} C_VEL
LIN {X 0,Y 488.808,Z 726.404,A -85,B 0,C 180,E1 -6671.612,E2 -6671.612} C_VEL
LIN {X 0,Y 488.764,Z 726.411,A -85,B 0,C 180,E1 -6675,E2 -6675} C_VEL
LIN {X 0,Y 488.749,Z 726.407,A -85,B 0,C 180,E1 -6678.442,E2 -6678.442} C_VEL
LIN {X 0,Y 488.709,Z 726.424,A -85,B 0,C 180,E1 -6681.071,E2 -6681.071} C_VEL
LIN {X 0,Y 488.685,Z 726.418,A -85,B 0,C 180,E1 -6683.746,E2 -6683.746} C_VEL
LIN {X 0,Y 488.794,Z 726.405,A -85,B 0,C 180,E1 -6686.944,E2 -6686.944} C_VEL
LIN {X 0,Y 488.71,Z 726.417,A -85,B 0,C 180,E1 -6690.363,E2 -6690.363} C_VEL
LIN {X 0,Y 488.73,Z 726.415,A -85,B 0,C 180,E1 -6693.483,E2 -6693.483} C_VEL
LIN {X 0,Y 488.683,Z 726.42,A -85,B 0,C 180,E1 -6696.354,E2 -6696.354} C_VEL
LIN {X 0,Y 488.702,Z 726.421,A -85,B 0,C 180,E1 -6699.254,E2 -6699.254} C_VEL
LIN {X 0,Y 488.708,Z 726.401,A -85,B 0,C 180,E1 -6701.6,E2 -6701.6} C_VEL
LIN {X 0,Y 488.702,Z 726.411,A -85,B 0,C 180,E1 -6704.803,E2 -6704.803} C_VEL
LIN {X 0,Y 488.693,Z 726.428,A -85,B 0,C 180,E1 -6707.475,E2 -6707.475} C_VEL
LIN {X 0,Y 488.735,Z 726.414,A -85,B 0,C 180,E1 -6709.677,E2 -6709.677} C_VEL
LIN {X 0,Y 488.68,Z 726.415,A -85,B 0,C 180,E1 -6712.841,E2 -6712.841} C_VEL
LIN {X 0,Y 488.725,Z 726.42,A -85,B 0,C 180,E1 -6715.887,E2 -6715.887} C_VEL
LIN {X 0,Y 488.692,Z 726.414,A -85,B 0,C 180,E1 -6718.82,E2 -6718.82} C_VEL
LIN {X 0,Y 488.714,Z 726.424,A -85,B 0,C 180,E1 -6721.669,E2 -6721.669} C_VEL
LIN {X 0,Y 488.704,Z 726.42,A -85,B 0,C 180,E1 -6724.341,E2 -6724.341} C_VEL
LIN {X 0,Y 488.063,Z 726.502,A -85,B 0,C 180,E1 -6725.029,E2 -6725.029} C_VEL
LIN {X 0,Y 485.211,Z 726.861,A -85,B 0,C 180,E1 -6726.146,E2 -6726.146} C_VEL
LIN {X 0,Y 482.777,Z 727.163,A -85,B 0,C 180,E1 -6727.046,E2 -6727.046} C_VEL
LIN {X 0,Y 481.725,Z 727.293,A -85,B 0,C 180,E1 -6727.742,E2 -6727.742} C_VEL
LIN {X 0,Y 481.637,Z 727.301,A -85,B 0,C 180,E1 -6727.977,E2 -6727.977} C_VEL
LIN {X 0,Y 481.793,Z 727.405,A -85,B 0,C 180,E1 -6730.784,E2 -6730.784} C_VEL
LIN {X 0,Y 482.136,Z 731.144,A -85,B 0,C 180,E1 -6731.773,E2 -6731.773} C_VEL
LIN {X 0,Y 481.817,Z 743.121,A -85,B 0,C 180,E1 -6734.778,E2 -6734.778} C_VEL
LIN {X 0,Y 481.558,Z 752.584,A -85,B 0,C 180,E1 -6737.046,E2 -6737.046} C_VEL
LIN {X 0,Y 482.213,Z 756.835,A -85,B 0,C 180,E1 -6737.173,E2 -6737.173} C_VEL
LIN {X 0,Y 483.378,Z 764.343,A -85,B 0,C 180,E1 -6737.317,E2 -6737.317} C_VEL
LIN {X 0,Y 483.079,Z 827.658,A -85,B 0,C 180,E1 -6738.275,E2 -6738.275} C_VEL
LIN {X 0,Y 482.971,Z 836.778,A -85,B 0,C 180,E1 -6738.511,E2 -6738.511} C_VEL
LIN {X 0,Y 482.745,Z 846.38,A -85,B 0,C 180,E1 -6738.878,E2 -6738.878} C_VEL
LIN {X 0,Y 482.547,Z 856.421,A -85,B 0,C 180,E1 -6739.404,E2 -6739.404} C_VEL
LIN {X 0,Y 482.192,Z 866.841,A -85,B 0,C 180,E1 -6740.139,E2 -6740.139} C_VEL
LIN {X 0,Y 481.915,Z 874.981,A -85,B 0,C 180,E1 -6740.875,E2 -6740.875} C_VEL
LIN {X 0,Y 481.643,Z 881.696,A -85,B 0,C 180,E1 -6741.61,E2 -6741.61} C_VEL
LIN {X 0,Y 481.417,Z 888.051,A -85,B 0,C 180,E1 -6742.45,E2 -6742.45} C_VEL
LIN {X 0,Y 481.289,Z 893.331,A -85,B 0,C 180,E1 -6743.291,E2 -6743.291} C_VEL
LIN {X 0,Y 481.208,Z 897.738,A -85,B 0,C 180,E1 -6744.132,E2 -6744.132} C_VEL
LIN {X 0,Y 480.945,Z 901.415,A -85,B 0,C 180,E1 -6744.97,E2 -6744.97} C_VEL
LIN {X 0,Y 481.025,Z 904.406,A -85,B 0,C 180,E1 -6745.811,E2 -6745.811} C_VEL
LIN {X 0,Y 480.921,Z 906.729,A -85,B 0,C 180,E1 -6746.649,E2 -6746.649} C_VEL
LIN {X 0,Y 480.849,Z 908.5,A -85,B 0,C 180,E1 -6747.487,E2 -6747.487} C_VEL
LIN {X 0,Y 480.822,Z 909.777,A -85,B 0,C 180,E1 -6748.325,E2 -6748.325} C_VEL
LIN {X 0,Y 480.757,Z 910.586,A -85,B 0,C 180,E1 -6749.162,E2 -6749.162} C_VEL
LIN {X 0,Y 480.741,Z 910.894,A -85,B 0,C 180,E1 -6750,E2 -6750} C_VEL
LIN {X 0,Y 480.758,Z 910.621,A -85,B 0,C 180,E1 -6750.838,E2 -6750.838} C_VEL
LIN {X 0,Y 480.823,Z 909.88,A -85,B 0,C 180,E1 -6751.675,E2 -6751.675} C_VEL
LIN {X 0,Y 480.849,Z 908.674,A -85,B 0,C 180,E1 -6752.513,E2 -6752.513} C_VEL
LIN {X 0,Y 480.97,Z 905.83,A -85,B 0,C 180,E1 -6753.77,E2 -6753.77} C_VEL
LIN {X 0,Y 480.991,Z 903.246,A -85,B 0,C 180,E1 -6754.609,E2 -6754.609} C_VEL
LIN {X 0,Y 481.192,Z 898.149,A -85,B 0,C 180,E1 -6755.868,E2 -6755.868} C_VEL
LIN {X 0,Y 481.272,Z 892.786,A -85,B 0,C 180,E1 -6756.898,E2 -6756.898} C_VEL
LIN {X 0,Y 481.516,Z 885.785,A -85,B 0,C 180,E1 -6757.97,E2 -6757.97} C_VEL
LIN {X 0,Y 481.793,Z 877.877,A -85,B 0,C 180,E1 -6758.916,E2 -6758.916} C_VEL
LIN {X 0,Y 482.099,Z 870.332,A -85,B 0,C 180,E1 -6759.651,E2 -6759.651} C_VEL
LIN {X 0,Y 482.303,Z 862.429,A -85,B 0,C 180,E1 -6760.283,E2 -6760.283} C_VEL
LIN {X 0,Y 482.578,Z 854.267,A -85,B 0,C 180,E1 -6760.807,E2 -6760.807} C_VEL
LIN {X 0,Y 482.819,Z 846.004,A -85,B 0,C 180,E1 -6761.227,E2 -6761.227} C_VEL
LIN {X 0,Y 482.96,Z 837.094,A -85,B 0,C 180,E1 -6761.569,E2 -6761.569} C_VEL
LIN {X 0,Y 483.113,Z 827.793,A -85,B 0,C 180,E1 -6761.812,E2 -6761.812} C_VEL
LIN {X 0,Y 483.274,Z 763.505,A -85,B 0,C 180,E1 -6762.788,E2 -6762.788} C_VEL
LIN {X 0,Y 481.533,Z 752.58,A -85,B 0,C 180,E1 -6763,E2 -6763} C_VEL
LIN {X 0,Y 481.889,Z 740.015,A -85,B 0,C 180,E1 -6766.087,E2 -6766.087} C_VEL
LIN {X 0,Y 482.105,Z 729.891,A -85,B 0,C 180,E1 -6768.638,E2 -6768.638} C_VEL
LIN {X 0,Y 481.753,Z 727.384,A -85,B 0,C 180,E1 -6769.328,E2 -6769.328} C_VEL
LIN {X 0,Y 481.65,Z 727.303,A -85,B 0,C 180,E1 -6772.295,E2 -6772.295} C_VEL
LIN {X 0,Y 481.67,Z 727.296,A -85,B 0,C 180,E1 -6775.225,E2 -6775.225} C_VEL
LIN {X 0,Y 481.662,Z 727.298,A -85,B 0,C 180,E1 -6777.834,E2 -6777.834} C_VEL
LIN {X 0,Y 481.645,Z 727.296,A -85,B 0,C 180,E1 -6780.711,E2 -6780.711} C_VEL
LIN {X 0,Y 481.676,Z 727.294,A -85,B 0,C 180,E1 -6783.729,E2 -6783.729} C_VEL
LIN {X 0,Y 481.627,Z 727.299,A -85,B 0,C 180,E1 -6786.747,E2 -6786.747} C_VEL
LIN {X 0,Y 481.677,Z 727.287,A -85,B 0,C 180,E1 -6789.94,E2 -6789.94} C_VEL
LIN {X 0,Y 481.639,Z 727.298,A -85,B 0,C 180,E1 -6793.3,E2 -6793.3} C_VEL
LIN {X 0,Y 481.654,Z 727.288,A -85,B 0,C 180,E1 -6795.641,E2 -6795.641} C_VEL
LIN {X 0,Y 481.657,Z 727.288,A -85,B 0,C 180,E1 -6798.958,E2 -6798.958} C_VEL
LIN {X 0,Y 481.655,Z 727.295,A -85,B 0,C 180,E1 -6801.993,E2 -6801.993} C_VEL
LIN {X 0,Y 481.686,Z 727.29,A -85,B 0,C 180,E1 -6805.318,E2 -6805.318} C_VEL
LIN {X 0,Y 481.645,Z 727.295,A -85,B 0,C 180,E1 -6808.311,E2 -6808.311} C_VEL
LIN {X 0,Y 481.699,Z 727.293,A -85,B 0,C 180,E1 -6811.218,E2 -6811.218} C_VEL
LIN {X 0,Y 481.698,Z 727.281,A -85,B 0,C 180,E1 -6814.043,E2 -6814.043} C_VEL
LIN {X 0,Y 481.676,Z 727.295,A -85,B 0,C 180,E1 -6816.812,E2 -6816.812} C_VEL
LIN {X 0,Y 481.697,Z 727.292,A -85,B 0,C 180,E1 -6819.503,E2 -6819.503} C_VEL
LIN {X 0,Y 481.694,Z 727.282,A -85,B 0,C 180,E1 -6822.158,E2 -6822.158} C_VEL
LIN {X 0,Y 481.746,Z 727.281,A -85,B 0,C 180,E1 -6824.776,E2 -6824.776} C_VEL
LIN {X 0,Y 481.753,Z 727.283,A -85,B 0,C 180,E1 -6828.215,E2 -6828.215} C_VEL
LIN {X 0,Y 481.763,Z 727.275,A -85,B 0,C 180,E1 -6831.612,E2 -6831.612} C_VEL
LIN {X 0,Y 481.811,Z 727.272,A -85,B 0,C 180,E1 -6834.139,E2 -6834.139} C_VEL
LIN {X 0,Y 481.931,Z 727.269,A -85,B 0,C 180,E1 -6837.492,E2 -6837.492} C_VEL
LIN {X 0,Y 481.943,Z 727.257,A -85,B 0,C 180,E1 -6840,E2 -6840} C_VEL
LIN {X 0,Y 481.93,Z 727.249,A -85,B 0,C 180,E1 -6842.507,E2 -6842.507} C_VEL
LIN {X 0,Y 481.812,Z 727.281,A -85,B 0,C 180,E1 -6845.86,E2 -6845.86} C_VEL
LIN {X 0,Y 481.765,Z 727.282,A -85,B 0,C 180,E1 -6848.388,E2 -6848.388} C_VEL
LIN {X 0,Y 481.753,Z 727.28,A -85,B 0,C 180,E1 -6851.785,E2 -6851.785} C_VEL
LIN {X 0,Y 481.745,Z 727.283,A -85,B 0,C 180,E1 -6855.224,E2 -6855.224} C_VEL
LIN {X 0,Y 481.715,Z 727.286,A -85,B 0,C 180,E1 -6858.722,E2 -6858.722} C_VEL
LIN {X 0,Y 481.649,Z 727.289,A -85,B 0,C 180,E1 -6861.394,E2 -6861.394} C_VEL
LIN {X 0,Y 481.679,Z 727.3,A -85,B 0,C 180,E1 -6864.113,E2 -6864.113} C_VEL
LIN {X 0,Y 481.749,Z 727.283,A -85,B 0,C 180,E1 -6867.139,E2 -6867.139} C_VEL
LIN {X 0,Y 481.68,Z 727.289,A -85,B 0,C 180,E1 -6869.741,E2 -6869.741} C_VEL
LIN {X 0,Y 481.674,Z 727.296,A -85,B 0,C 180,E1 -6872.674,E2 -6872.674} C_VEL
LIN {X 0,Y 481.645,Z 727.296,A -85,B 0,C 180,E1 -6875.709,E2 -6875.709} C_VEL
LIN {X 0,Y 481.715,Z 727.263,A -85,B 0,C 180,E1 -6879.354,E2 -6879.354} C_VEL
LIN {X 0,Y 481.65,Z 727.292,A -85,B 0,C 180,E1 -6882.16,E2 -6882.16} C_VEL
LIN {X 0,Y 481.66,Z 727.295,A -85,B 0,C 180,E1 -6885.543,E2 -6885.543} C_VEL
LIN {X 0,Y 481.658,Z 727.293,A -85,B 0,C 180,E1 -6888.958,E2 -6888.958} C_VEL
LIN {X 0,Y 481.673,Z 727.295,A -85,B 0,C 180,E1 -6891.141,E2 -6891.141} C_VEL
LIN {X 0,Y 481.669,Z 727.299,A -85,B 0,C 180,E1 -6894.795,E2 -6894.795} C_VEL
LIN {X 0,Y 481.674,Z 727.292,A -85,B 0,C 180,E1 -6897.326,E2 -6897.326} C_VEL
LIN {X 0,Y 481.68,Z 727.288,A -85,B 0,C 180,E1 -6900.259,E2 -6900.259} C_VEL
LIN {X 0,Y 481.746,Z 727.283,A -85,B 0,C 180,E1 -6903.112,E2 -6903.112} C_VEL
LIN {X 0,Y 481.68,Z 727.294,A -85,B 0,C 180,E1 -6906.345,E2 -6906.345} C_VEL
LIN {X 0,Y 481.743,Z 727.6,A -85,B 0,C 180,E1 -6906.65,E2 -6906.65} C_VEL
LIN {X 0,Y 482.962,Z 735.098,A -85,B 0,C 180,E1 -6908.263,E2 -6908.263} C_VEL
LIN {X 0,Y 482.478,Z 749.765,A -85,B 0,C 180,E1 -6911.23,E2 -6911.23} C_VEL
LIN {X 0,Y 481.967,Z 764.849,A -85,B 0,C 180,E1 -6914.24,E2 -6914.24} C_VEL
LIN {X 0,Y 481.618,Z 778.829,A -85,B 0,C 180,E1 -6916.98,E2 -6916.98} C_VEL
LIN {X 0,Y 481.975,Z 781.737,A -85,B 0,C 180,E1 -6917.08,E2 -6917.08} C_VEL
LIN {X 0,Y 483.356,Z 793.296,A -85,B 0,C 180,E1 -6917.289,E2 -6917.289} C_VEL
LIN {X 0,Y 483.061,Z 856.383,A -85,B 0,C 180,E1 -6918.247,E2 -6918.247} C_VEL
LIN {X 0,Y 482.8,Z 866.858,A -85,B 0,C 180,E1 -6918.534,E2 -6918.534} C_VEL
LIN {X 0,Y 482.59,Z 877.579,A -85,B 0,C 180,E1 -6918.981,E2 -6918.981} C_VEL
LIN {X 0,Y 482.271,Z 888.214,A -85,B 0,C 180,E1 -6919.611,E2 -6919.611} C_VEL
LIN {X 0,Y 482.009,Z 896.544,A -85,B 0,C 180,E1 -6920.241,E2 -6920.241} C_VEL
LIN {X 0,Y 481.731,Z 904.427,A -85,B 0,C 180,E1 -6920.977,E2 -6920.977} C_VEL
LIN {X 0,Y 481.458,Z 911.798,A -85,B 0,C 180,E1 -6921.818,E2 -6921.818} C_VEL
LIN {X 0,Y 481.265,Z 919.279,A -85,B 0,C 180,E1 -6922.87,E2 -6922.87} C_VEL
LIN {X 0,Y 481.093,Z 926.111,A -85,B 0,C 180,E1 -6924.131,E2 -6924.131} C_VEL
LIN {X 0,Y 480.896,Z 931.294,A -85,B 0,C 180,E1 -6925.39,E2 -6925.39} C_VEL
LIN {X 0,Y 480.917,Z 935.105,A -85,B 0,C 180,E1 -6926.649,E2 -6926.649} C_VEL
LIN {X 0,Y 480.806,Z 936.855,A -85,B 0,C 180,E1 -6927.487,E2 -6927.487} C_VEL
LIN {X 0,Y 480.788,Z 938.111,A -85,B 0,C 180,E1 -6928.325,E2 -6928.325} C_VEL
LIN {X 0,Y 480.757,Z 938.892,A -85,B 0,C 180,E1 -6929.162,E2 -6929.162} C_VEL
LIN {X 0,Y 480.74,Z 939.187,A -85,B 0,C 180,E1 -6930,E2 -6930} C_VEL
LIN {X 0,Y 480.757,Z 938.891,A -85,B 0,C 180,E1 -6930.838,E2 -6930.838} C_VEL
LIN {X 0,Y 480.788,Z 938.11,A -85,B 0,C 180,E1 -6931.675,E2 -6931.675} C_VEL
LIN {X 0,Y 480.806,Z 936.854,A -85,B 0,C 180,E1 -6932.513,E2 -6932.513} C_VEL
LIN {X 0,Y 480.944,Z 933.948,A -85,B 0,C 180,E1 -6933.77,E2 -6933.77} C_VEL
LIN {X 0,Y 480.896,Z 931.294,A -85,B 0,C 180,E1 -6934.61,E2 -6934.61} C_VEL
LIN {X 0,Y 481.093,Z 926.108,A -85,B 0,C 180,E1 -6935.869,E2 -6935.869} C_VEL
LIN {X 0,Y 481.26,Z 919.272,A -85,B 0,C 180,E1 -6937.13,E2 -6937.13} C_VEL
LIN {X 0,Y 481.458,Z 911.8,A -85,B 0,C 180,E1 -6938.182,E2 -6938.182} C_VEL
LIN {X 0,Y 481.731,Z 904.433,A -85,B 0,C 180,E1 -6939.023,E2 -6939.023} C_VEL
LIN {X 0,Y 482.009,Z 896.547,A -85,B 0,C 180,E1 -6939.759,E2 -6939.759} C_VEL
LIN {X 0,Y 482.271,Z 888.215,A -85,B 0,C 180,E1 -6940.389,E2 -6940.389} C_VEL
LIN {X 0,Y 482.605,Z 877.583,A -85,B 0,C 180,E1 -6941.019,E2 -6941.019} C_VEL
LIN {X 0,Y 482.834,Z 866.03,A -85,B 0,C 180,E1 -6941.492,E2 -6941.492} C_VEL
LIN {X 0,Y 483.055,Z 856.384,A -85,B 0,C 180,E1 -6941.753,E2 -6941.753} C_VEL
LIN {X 0,Y 483.264,Z 814.383,A -85,B 0,C 180,E1 -6942.399,E2 -6942.399} C_VEL
LIN {X 0,Y 483.217,Z 791.332,A -85,B 0,C 180,E1 -6942.744,E2 -6942.744} C_VEL
LIN {X 0,Y 481.617,Z 779.102,A -85,B 0,C 180,E1 -6942.994,E2 -6942.994} C_VEL
LIN {X 0,Y 481.792,Z 771.885,A -85,B 0,C 180,E1 -6944.358,E2 -6944.358} C_VEL
LIN {X 0,Y 482.248,Z 756.693,A -85,B 0,C 180,E1 -6947.383,E2 -6947.383} C_VEL
LIN {X 0,Y 482.836,Z 740.341,A -85,B 0,C 180,E1 -6950.669,E2 -6950.669} C_VEL
LIN {X 0,Y 482.846,Z 733.779,A -85,B 0,C 180,E1 -6952.012,E2 -6952.012} C_VEL
LIN {X 0,Y 481.697,Z 727.338,A -85,B 0,C 180,E1 -6953.451,E2 -6953.451} C_VEL
LIN {X 0,Y 481.701,Z 727.29,A -85,B 0,C 180,E1 -6955.957,E2 -6955.957} C_VEL
LIN {X 0,Y 481.701,Z 727.295,A -85,B 0,C 180,E1 -6958.781,E2 -6958.781} C_VEL
LIN {X 0,Y 481.66,Z 727.294,A -85,B 0,C 180,E1 -6962.19,E2 -6962.19} C_VEL
LIN {X 0,Y 481.694,Z 727.293,A -85,B 0,C 180,E1 -6964.682,E2 -6964.682} C_VEL
LIN {X 0,Y 481.658,Z 727.298,A -85,B 0,C 180,E1 -6968.008,E2 -6968.008} C_VEL
LIN {X 0,Y 481.663,Z 727.289,A -85,B 0,C 180,E1 -6970.647,E2 -6970.647} C_VEL
LIN {X 0,Y 481.64,Z 727.298,A -85,B 0,C 180,E1 -6973.3,E2 -6973.3} C_VEL
LIN {X 0,Y 481.659,Z 727.302,A -85,B 0,C 180,E1 -6975.641,E2 -6975.641} C_VEL
LIN {X 0,Y 481.669,Z 727.284,A -85,B 0,C 180,E1 -6978.96,E2 -6978.96} C_VEL
LIN {X 0,Y 481.699,Z 727.266,A -85,B 0,C 180,E1 -6981.144,E2 -6981.144} C_VEL
LIN {X 0,Y 481.67,Z 727.291,A -85,B 0,C 180,E1 -6984.795,E2 -6984.795} C_VEL
LIN {X 0,Y 481.674,Z 727.296,A -85,B 0,C 180,E1 -6987.326,E2 -6987.326} C_VEL
LIN {X 0,Y 481.68,Z 727.289,A -85,B 0,C 180,E1 -6990.259,E2 -6990.259} C_VEL
LIN {X 0,Y 481.747,Z 727.283,A -85,B 0,C 180,E1 -6993.112,E2 -6993.112} C_VEL
LIN {X 0,Y 481.679,Z 727.299,A -85,B 0,C 180,E1 -6995.887,E2 -6995.887} C_VEL
LIN {X 0,Y 481.704,Z 727.281,A -85,B 0,C 180,E1 -6999.028,E2 -6999.028} C_VEL
LIN {X 0,Y 481.71,Z 727.296,A -85,B 0,C 180,E1 -7002.159,E2 -7002.159} C_VEL
LIN {X 0,Y 481.745,Z 727.283,A -85,B 0,C 180,E1 -7004.776,E2 -7004.776} C_VEL
LIN {X 0,Y 481.753,Z 727.279,A -85,B 0,C 180,E1 -7008.215,E2 -7008.215} C_VEL
LIN {X 0,Y 481.765,Z 727.282,A -85,B 0,C 180,E1 -7011.612,E2 -7011.612} C_VEL
LIN {X 0,Y 481.812,Z 727.281,A -85,B 0,C 180,E1 -7014.14,E2 -7014.14} C_VEL
LIN {X 0,Y 481.931,Z 727.249,A -85,B 0,C 180,E1 -7017.493,E2 -7017.493} C_VEL
LIN {X 0,Y 481.908,Z 727.268,A -85,B 0,C 180,E1 -7020.836,E2 -7020.836} C_VEL
LIN {X 0,Y 481.931,Z 727.269,A -85,B 0,C 180,E1 -7022.508,E2 -7022.508} C_VEL
LIN {X 0,Y 481.811,Z 727.272,A -85,B 0,C 180,E1 -7025.861,E2 -7025.861} C_VEL
LIN {X 0,Y 481.764,Z 727.274,A -85,B 0,C 180,E1 -7028.388,E2 -7028.388} C_VEL
LIN {X 0,Y 481.753,Z 727.283,A -85,B 0,C 180,E1 -7031.785,E2 -7031.785} C_VEL
LIN {X 0,Y 481.745,Z 727.282,A -85,B 0,C 180,E1 -7035.224,E2 -7035.224} C_VEL
LIN {X 0,Y 481.71,Z 727.287,A -85,B 0,C 180,E1 -7038.722,E2 -7038.722} C_VEL
LIN {X 0,Y 481.647,Z 727.299,A -85,B 0,C 180,E1 -7041.395,E2 -7041.395} C_VEL
LIN {X 0,Y 481.67,Z 727.291,A -85,B 0,C 180,E1 -7044.114,E2 -7044.114} C_VEL
LIN {X 0,Y 481.748,Z 727.286,A -85,B 0,C 180,E1 -7047.139,E2 -7047.139} C_VEL
LIN {X 0,Y 481.68,Z 727.294,A -85,B 0,C 180,E1 -7049.741,E2 -7049.741} C_VEL
LIN {X 0,Y 481.672,Z 727.292,A -85,B 0,C 180,E1 -7052.674,E2 -7052.674} C_VEL
LIN {X 0,Y 481.637,Z 727.3,A -85,B 0,C 180,E1 -7055.71,E2 -7055.71} C_VEL
LIN {X 0,Y 481.672,Z 727.295,A -85,B 0,C 180,E1 -7058.859,E2 -7058.859} C_VEL
LIN {X 0,Y 481.653,Z 727.274,A -85,B 0,C 180,E1 -7061.913,E2 -7061.913} C_VEL
LIN {X 0,Y 481.655,Z 727.287,A -85,B 0,C 180,E1 -7064.458,E2 -7064.458} C_VEL
LIN {X 0,Y 481.649,Z 727.3,A -85,B 0,C 180,E1 -7067.839,E2 -7067.839} C_VEL
LIN {X 0,Y 481.662,Z 727.288,A -85,B 0,C 180,E1 -7070.654,E2 -7070.654} C_VEL
LIN {X 0,Y 481.629,Z 727.299,A -85,B 0,C 180,E1 -7073.376,E2 -7073.376} C_VEL
LIN {X 0,Y 481.678,Z 727.294,A -85,B 0,C 180,E1 -7076.327,E2 -7076.327} C_VEL
LIN {X 0,Y 481.65,Z 727.296,A -85,B 0,C 180,E1 -7079.418,E2 -7079.418} C_VEL
LIN {X 0,Y 481.669,Z 727.298,A -85,B 0,C 180,E1 -7082.166,E2 -7082.166} C_VEL
LIN {X 0,Y 481.678,Z 727.294,A -85,B 0,C 180,E1 -7084.968,E2 -7084.968} C_VEL
LIN {X 0,Y 481.637,Z 727.301,A -85,B 0,C 180,E1 -7087.977,E2 -7087.977} C_VEL
LIN {X 0,Y 480.957,Z 727.386,A -85,B 0,C 180,E1 -7088.443,E2 -7088.443} C_VEL
LIN {X 0,Y 475.327,Z 728.094,A -85,B 0,C 180,E1 -7089.912,E2 -7089.912} C_VEL
LIN {X 0,Y 474.695,Z 728.188,A -85,B 0,C 180,E1 -7090.387,E2 -7090.387} C_VEL
LIN {X 0,Y 474.769,Z 728.381,A -85,B 0,C 180,E1 -7090.713,E2 -7090.713} C_VEL
LIN {X 0,Y 475.109,Z 732.888,A -85,B 0,C 180,E1 -7091.902,E2 -7091.902} C_VEL
LIN {X 0,Y 474.747,Z 745.033,A -85,B 0,C 180,E1 -7094.985,E2 -7094.985} C_VEL
LIN {X 0,Y 474.527,Z 752.677,A -85,B 0,C 180,E1 -7096.836,E2 -7096.836} C_VEL
LIN {X 0,Y 474.821,Z 754.713,A -85,B 0,C 180,E1 -7096.933,E2 -7096.933} C_VEL
LIN {X 0,Y 476.443,Z 764.603,A -85,B 0,C 180,E1 -7097.129,E2 -7097.129} C_VEL
LIN {X 0,Y 476.153,Z 827.898,A -85,B 0,C 180,E1 -7098.102,E2 -7098.102} C_VEL
LIN {X 0,Y 476.047,Z 837.007,A -85,B 0,C 180,E1 -7098.342,E2 -7098.342} C_VEL
LIN {X 0,Y 475.81,Z 846.603,A -85,B 0,C 180,E1 -7098.714,E2 -7098.714} C_VEL
LIN {X 0,Y 475.578,Z 856.641,A -85,B 0,C 180,E1 -7099.247,E2 -7099.247} C_VEL
LIN {X 0,Y 475.196,Z 867.058,A -85,B 0,C 180,E1 -7099.992,E2 -7099.992} C_VEL
LIN {X 0,Y 474.924,Z 875.196,A -85,B 0,C 180,E1 -7100.739,E2 -7100.739} C_VEL
LIN {X 0,Y 474.619,Z 881.91,A -85,B 0,C 180,E1 -7101.485,E2 -7101.485} C_VEL
LIN {X 0,Y 474.395,Z 888.263,A -85,B 0,C 180,E1 -7102.338,E2 -7102.338} C_VEL
LIN {X 0,Y 474.222,Z 893.544,A -85,B 0,C 180,E1 -7103.191,E2 -7103.191} C_VEL
LIN {X 0,Y 474.17,Z 897.949,A -85,B 0,C 180,E1 -7104.045,E2 -7104.045} C_VEL
LIN {X 0,Y 473.884,Z 901.626,A -85,B 0,C 180,E1 -7104.895,E2 -7104.895} C_VEL
LIN {X 0,Y 473.933,Z 904.618,A -85,B 0,C 180,E1 -7105.748,E2 -7105.748} C_VEL
LIN {X 0,Y 473.855,Z 906.939,A -85,B 0,C 180,E1 -7106.599,E2 -7106.599} C_VEL
LIN {X 0,Y 473.766,Z 908.71,A -85,B 0,C 180,E1 -7107.449,E2 -7107.449} C_VEL
LIN {X 0,Y 473.726,Z 909.986,A -85,B 0,C 180,E1 -7108.3,E2 -7108.3} C_VEL
LIN {X 0,Y 473.686,Z 910.795,A -85,B 0,C 180,E1 -7109.15,E2 -7109.15} C_VEL
LIN {X 0,Y 473.668,Z 911.103,A -85,B 0,C 180,E1 -7110,E2 -7110} C_VEL
LIN {X 0,Y 473.687,Z 910.829,A -85,B 0,C 180,E1 -7110.85,E2 -7110.85} C_VEL
LIN {X 0,Y 473.727,Z 910.088,A -85,B 0,C 180,E1 -7111.7,E2 -7111.7} C_VEL
LIN {X 0,Y 473.766,Z 908.881,A -85,B 0,C 180,E1 -7112.551,E2 -7112.551} C_VEL
LIN {X 0,Y 473.906,Z 906.037,A -85,B 0,C 180,E1 -7113.826,E2 -7113.826} C_VEL
LIN {X 0,Y 473.896,Z 903.453,A -85,B 0,C 180,E1 -7114.679,E2 -7114.679} C_VEL
LIN {X 0,Y 474.15,Z 898.354,A -85,B 0,C 180,E1 -7115.956,E2 -7115.956} C_VEL
LIN {X 0,Y 474.289,Z 891.664,A -85,B 0,C 180,E1 -7117.236,E2 -7117.236} C_VEL
LIN {X 0,Y 474.537,Z 884.316,A -85,B 0,C 180,E1 -7118.303,E2 -7118.303} C_VEL
LIN {X 0,Y 474.838,Z 877.061,A -85,B 0,C 180,E1 -7119.155,E2 -7119.155} C_VEL
LIN {X 0,Y 475.102,Z 870.533,A -85,B 0,C 180,E1 -7119.795,E2 -7119.795} C_VEL
LIN {X 0,Y 475.325,Z 862.628,A -85,B 0,C 180,E1 -7120.435,E2 -7120.435} C_VEL
LIN {X 0,Y 475.622,Z 854.463,A -85,B 0,C 180,E1 -7120.967,E2 -7120.967} C_VEL
LIN {X 0,Y 475.877,Z 846.197,A -85,B 0,C 180,E1 -7121.393,E2 -7121.393} C_VEL
LIN {X 0,Y 476.033,Z 837.282,A -85,B 0,C 180,E1 -7121.739,E2 -7121.739} C_VEL
LIN {X 0,Y 476.192,Z 828.09,A -85,B 0,C 180,E1 -7121.983,E2 -7121.983} C_VEL
LIN {X 0,Y 476.39,Z 764.328,A -85,B 0,C 180,E1 -7122.966,E2 -7122.966} C_VEL
LIN {X 0,Y 474.512,Z 752.747,A -85,B 0,C 180,E1 -7123.196,E2 -7123.196} C_VEL
LIN {X 0,Y 474.884,Z 740.174,A -85,B 0,C 180,E1 -7126.331,E2 -7126.331} C_VEL
LIN {X 0,Y 475.058,Z 730.653,A -85,B 0,C 180,E1 -7128.77,E2 -7128.77} C_VEL
LIN {X 0,Y 474.714,Z 728.25,A -85,B 0,C 180,E1 -7129.457,E2 -7129.457} C_VEL
LIN {X 0,Y 474.602,Z 728.177,A -85,B 0,C 180,E1 -7132.645,E2 -7132.645} C_VEL
LIN {X 0,Y 474.62,Z 728.174,A -85,B 0,C 180,E1 -7135.431,E2 -7135.431} C_VEL
LIN {X 0,Y 474.617,Z 728.178,A -85,B 0,C 180,E1 -7138.284,E2 -7138.284} C_VEL
